C09135=1233.030,93.308,-46.941,-178.457,5.464,148.489
C09136=1233.025,93.557,-46.959,-178.455,5.465,148.489
C09137=1233.020,93.807,-46.977,-178.453,5.466,148.488
C09138=1233.016,94.056,-46.996,-178.450,5.466,148.487
C09139=1233.011,94.305,-47.014,-178.448,5.467,148.487
C09140=1233.006,94.555,-47.032,-178.445,5.468,148.486
C09141=1233.001,94.804,-47.052,-178.442,5.469,148.486
C09142=1232.996,95.053,-47.070,-178.439,5.470,148.485
C09143=1232.991,95.302,-47.088,-178.437,5.471,148.485
C09144=1232.986,95.552,-47.107,-178.435,5.471,148.484
C09145=1232.982,95.801,-47.126,-178.432,5.472,148.483
C09146=1232.976,96.050,-47.145,-178.429,5.473,148.483
C09147=1232.972,96.299,-47.164,-178.427,5.474,148.482
C09148=1232.967,96.549,-47.182,-178.425,5.474,148.482
C09149=1232.962,96.799,-47.201,-178.422,5.475,148.481
C09150=1232.958,97.047,-47.219,-178.420,5.476,148.481
C09151=1232.953,97.296,-47.237,-178.417,5.477,148.480
C09152=1232.948,97.546,-47.257,-178.414,5.478,148.479
C09153=1232.943,97.795,-47.275,-178.412,5.478,148.479
C09154=1232.938,98.044,-47.294,-178.409,5.479,148.478
C09155=1232.934,98.293,-47.313,-178.407,5.480,148.478
C09156=1232.928,98.543,-47.332,-178.404,5.481,148.477
C09157=1232.924,98.792,-47.351,-178.402,5.481,148.476
C09158=1232.919,99.041,-47.369,-178.399,5.482,148.476
C09159=1232.914,99.290,-47.388,-178.396,5.484,148.475
C09160=1232.909,99.540,-47.407,-178.394,5.484,148.475
C09161=1232.904,99.789,-47.426,-178.392,5.485,148.474
C09162=1232.900,100.038,-47.445,-178.389,5.486,148.473
C09163=1232.894,100.288,-47.464,-178.386,5.486,148.473
C09164=1232.890,100.537,-47.483,-178.384,5.487,148.472
C09165=1232.885,100.786,-47.501,-178.382,5.488,148.472
C09166=1232.880,101.035,-47.520,-178.379,5.489,148.471
C09167=1232.875,101.284,-47.539,-178.376,5.490,148.470
C09168=1232.871,101.534,-47.557,-178.374,5.491,148.470
C09169=1232.866,101.783,-47.577,-178.371,5.492,148.469
C09170=1232.861,102.032,-47.596,-178.368,5.492,148.469
C09171=1232.856,102.282,-47.615,-178.366,5.493,148.468
C09172=1232.852,102.531,-47.633,-178.364,5.494,148.468
C09173=1232.847,102.780,-47.653,-178.361,5.495,148.467
C09174=1232.842,103.029,-47.671,-178.358,5.496,148.466
C09175=1232.837,103.278,-47.690,-178.356,5.497,148.466
C09176=1232.832,103.527,-47.709,-178.353,5.498,148.465
C09177=1232.827,103.776,-47.729,-178.351,5.498,148.465
C09178=1232.823,104.026,-47.747,-178.348,5.499,148.464
C09179=1232.817,104.275,-47.766,-178.346,5.500,148.464
C09180=1232.813,104.525,-47.786,-178.343,5.500,148.463
C09181=1232.808,104.773,-47.805,-178.340,5.502,148.463
C09182=1232.803,105.023,-47.824,-178.338,5.503,148.462
C09183=1232.798,105.272,-47.842,-178.335,5.503,148.461
C09184=1232.794,105.521,-47.862,-178.333,5.504,148.461
C09185=1232.788,105.770,-47.881,-178.331,5.505,148.460
C09186=1232.784,106.020,-47.900,-178.328,5.506,148.460
C09187=1232.779,106.269,-47.919,-178.325,5.507,148.459
C09188=1232.775,106.518,-47.938,-178.323,5.508,148.459
C09189=1232.769,106.767,-47.957,-178.320,5.509,148.458
C09190=1232.765,107.017,-47.977,-178.318,5.510,148.457
C09191=1232.761,107.266,-47.996,-178.315,5.510,148.457
C09192=1232.755,107.534,-48.017,-178.312,5.512,148.456
C09193=1232.750,107.803,-48.037,-178.309,5.512,148.456
C09194=1232.744,108.071,-48.058,-178.307,5.513,148.455
C09195=1232.739,108.340,-48.079,-178.304,5.514,148.454
C09196=1232.734,108.589,-48.098,-178.302,5.515,148.454
C09197=1232.730,108.838,-48.117,-178.299,5.516,148.453
C09198=1232.725,109.087,-48.137,-178.296,5.517,148.453
C09199=1232.720,109.337,-48.155,-178.294,5.518,148.452
C09200=1232.716,109.586,-48.175,-178.292,5.518,148.452
C09201=1232.710,109.835,-48.194,-178.288,5.520,148.451
C09202=1232.706,110.085,-48.213,-178.286,5.521,148.451
C09203=1232.701,110.333,-48.232,-178.284,5.521,148.450
C09204=1232.696,110.583,-48.252,-178.281,5.522,148.449
C09205=1232.692,110.832,-48.272,-178.279,5.523,148.449
C09206=1232.686,111.081,-48.291,-178.276,5.524,148.448
C09207=1232.682,111.330,-48.310,-178.273,5.525,148.448
C09208=1232.677,111.579,-48.329,-178.271,5.526,148.447
C09209=1232.672,111.829,-48.349,-178.268,5.527,148.446
C09210=1232.667,112.079,-48.368,-178.266,5.527,148.446
C09211=1232.663,112.327,-48.387,-178.264,5.528,148.445
C09212=1232.658,112.577,-48.407,-178.261,5.530,148.445
C09213=1232.653,112.825,-48.426,-178.258,5.531,148.444
C09214=1232.648,113.074,-48.446,-178.256,5.531,148.444
C09215=1232.644,113.324,-48.466,-178.253,5.532,148.443
C09216=1232.639,113.573,-48.485,-178.251,5.533,148.443
C09217=1232.634,113.822,-48.504,-178.248,5.534,148.442
C09218=1232.629,114.072,-48.524,-178.245,5.535,148.441
C09219=1232.624,114.321,-48.543,-178.243,5.536,148.441
C09220=1232.619,114.570,-48.563,-178.241,5.536,148.440
C09221=1232.615,114.819,-48.582,-178.238,5.537,148.440
C09222=1232.610,115.068,-48.601,-178.235,5.539,148.439
C09223=1232.606,115.317,-48.622,-178.233,5.540,148.439
C09224=1232.600,115.566,-48.641,-178.231,5.541,148.438
C09225=1232.595,115.816,-48.661,-178.228,5.541,148.438
C09226=1232.591,116.065,-48.680,-178.225,5.543,148.437
C09227=1232.585,116.314,-48.700,-178.223,5.544,148.437
C09228=1232.581,116.563,-48.719,-178.220,5.544,148.436
C09229=1232.577,116.812,-48.739,-178.217,5.545,148.435
C09230=1232.572,117.062,-48.759,-178.215,5.546,148.435
C09231=1232.567,117.311,-48.778,-178.212,5.547,148.434
C09232=1232.562,117.560,-48.798,-178.210,5.548,148.434
C09233=1232.557,117.810,-48.817,-178.207,5.549,148.433
C09234=1232.552,118.058,-48.837,-178.205,5.549,148.433
C09235=1232.548,118.308,-48.857,-178.202,5.551,148.432
C09236=1232.543,118.557,-48.877,-178.199,5.552,148.432
C09237=1232.538,118.805,-48.897,-178.197,5.553,148.431
C09238=1232.534,119.055,-48.916,-178.195,5.554,148.431
C09239=1232.529,119.304,-48.935,-178.192,5.554,148.430
C09240=1232.524,119.554,-48.955,-178.189,5.556,148.429
C09241=1232.519,119.802,-48.975,-178.187,5.557,148.429
C09242=1232.515,120.052,-48.995,-178.184,5.557,148.428
C09243=1232.510,120.301,-49.014,-178.182,5.558,148.428
C09244=1232.505,120.550,-49.035,-178.179,5.560,148.427
C09245=1232.500,120.799,-49.054,-178.177,5.561,148.427
C09246=1232.495,121.049,-49.074,-178.174,5.561,148.426
C09247=1232.491,121.298,-49.094,-178.172,5.562,148.425
C09248=1232.486,121.547,-49.114,-178.169,5.564,148.425
C09249=1232.481,121.795,-49.134,-178.166,5.564,148.424
C09250=1232.476,122.045,-49.153,-178.164,5.565,148.424
C09251=1232.472,122.295,-49.173,-178.162,5.566,148.423
C09252=1232.467,122.543,-49.193,-178.158,5.567,148.423
C09253=1232.462,122.792,-49.213,-178.156,5.568,148.422
C09254=1232.457,123.041,-49.233,-178.154,5.569,148.422
C09255=1232.453,123.291,-49.253,-178.152,5.570,148.421
C09256=1232.448,123.540,-49.272,-178.148,5.571,148.421
C09257=1232.443,123.789,-49.293,-178.146,5.572,148.420
C09258=1232.438,124.038,-49.312,-178.144,5.573,148.420
C09259=1232.433,124.288,-49.333,-178.141,5.574,148.419
C09260=1232.428,124.537,-49.353,-178.138,5.576,148.419
C09261=1232.424,124.786,-49.373,-178.136,5.576,148.418
C09262=1232.419,125.036,-49.393,-178.133,5.577,148.417
C09263=1232.414,125.284,-49.413,-178.131,5.578,148.417
C09264=1232.409,125.533,-49.432,-178.128,5.579,148.416
C09265=1232.405,125.782,-49.453,-178.126,5.580,148.416
C09266=1232.400,126.032,-49.472,-178.123,5.581,148.415
C09267=1232.396,126.281,-49.493,-178.121,5.583,148.415
C09268=1232.391,126.530,-49.513,-178.118,5.583,148.414
C09269=1232.385,126.779,-49.533,-178.115,5.584,148.414
C09270=1232.381,127.028,-49.553,-178.113,5.585,148.413
C09271=1232.376,127.278,-49.573,-178.110,5.586,148.413
C09272=1232.371,127.526,-49.593,-178.108,5.587,148.412
C09273=1232.367,127.775,-49.614,-178.105,5.588,148.412
C09274=1232.362,128.025,-49.633,-178.103,5.589,148.411
C09275=1232.358,128.274,-49.654,-178.100,5.590,148.411
C09276=1232.352,128.524,-49.674,-178.097,5.591,148.410
C09277=1232.347,128.772,-49.694,-178.095,5.592,148.410
C09278=1232.343,129.021,-49.714,-178.092,5.594,148.409
C09279=1232.338,129.271,-49.734,-178.090,5.595,148.409
C09280=1232.334,129.520,-49.755,-178.087,5.595,148.408
C09281=1232.329,129.769,-49.775,-178.085,5.596,148.407
C09282=1232.324,130.018,-49.795,-178.082,5.598,148.407
C09283=1232.319,130.267,-49.816,-178.080,5.599,148.406
C09284=1232.315,130.516,-49.836,-178.077,5.599,148.406
C09285=1232.310,130.765,-49.856,-178.074,5.601,148.405
C09286=1232.304,131.014,-49.876,-178.072,5.602,148.405
C09287=1232.300,131.263,-49.897,-178.070,5.602,148.404
C09288=1232.295,131.512,-49.917,-178.067,5.604,148.404
C09289=1232.291,131.762,-49.937,-178.064,5.605,148.403
C09290=1232.286,132.011,-49.958,-178.062,5.606,148.403
C09291=1232.281,132.260,-49.978,-178.060,5.606,148.402
C09292=1232.277,132.509,-49.998,-178.057,5.608,148.402
C09293=1232.272,132.758,-50.019,-178.054,5.609,148.401
C09294=1232.267,133.008,-50.039,-178.052,5.610,148.400
C09295=1232.262,133.257,-50.059,-178.049,5.611,148.400
C09296=1232.257,133.525,-50.082,-178.046,5.612,148.399
C09297=1232.251,133.794,-50.103,-178.043,5.613,148.399
C09298=1232.247,134.063,-50.125,-178.041,5.614,148.398
C09299=1232.242,134.331,-50.148,-178.038,5.616,148.398
C09300=1232.237,134.581,-50.168,-178.035,5.617,148.397
C09301=1232.232,134.830,-50.189,-178.033,5.618,148.397
C09302=1232.228,135.079,-50.209,-178.030,5.619,148.396
C09303=1232.223,135.328,-50.229,-178.028,5.620,148.396
C09304=1232.218,135.577,-50.250,-178.025,5.621,148.395
C09305=1232.214,135.826,-50.271,-178.023,5.622,148.395
C09306=1232.209,136.075,-50.291,-178.020,5.623,148.394
C09307=1232.204,136.324,-50.312,-178.018,5.624,148.394
C09308=1232.200,136.573,-50.332,-178.015,5.626,148.393
C09309=1232.194,136.823,-50.353,-178.013,5.627,148.393
C09310=1232.190,137.071,-50.374,-178.010,5.627,148.392
C09311=1232.185,137.321,-50.393,-178.008,5.629,148.392
C09312=1232.180,137.570,-50.414,-178.005,5.630,148.391
C09313=1232.176,137.819,-50.435,-178.003,5.631,148.391
C09314=1232.170,138.069,-50.456,-178.000,5.632,148.390
C09315=1232.166,138.317,-50.476,-177.998,5.633,148.390
C09316=1232.161,138.567,-50.497,-177.995,5.634,148.389
C09317=1232.156,138.816,-50.517,-177.992,5.636,148.389
C09318=1232.152,139.065,-50.538,-177.990,5.636,148.388
C09319=1232.147,139.313,-50.559,-177.988,5.637,148.388
C09320=1232.143,139.562,-50.580,-177.984,5.639,148.387
C09321=1232.137,139.811,-50.601,-177.982,5.640,148.387
C09322=1232.133,140.060,-50.621,-177.980,5.640,148.386
C09323=1232.128,140.310,-50.642,-177.977,5.642,148.386
C09324=1232.123,140.559,-50.662,-177.974,5.643,148.385
C09325=1232.118,140.808,-50.683,-177.972,5.644,148.385
C09326=1232.114,141.057,-50.704,-177.969,5.645,148.384
C09327=1232.109,141.307,-50.725,-177.967,5.646,148.384
C09328=1232.105,141.556,-50.745,-177.964,5.647,148.383
C09329=1232.100,141.805,-50.766,-177.962,5.649,148.383
C09330=1232.095,142.053,-50.788,-177.959,5.649,148.382
C09331=1232.090,142.303,-50.808,-177.957,5.651,148.382
C09332=1232.086,142.552,-50.829,-177.954,5.652,148.381
C09333=1232.081,142.801,-50.850,-177.952,5.653,148.381
C09334=1232.076,143.050,-50.870,-177.949,5.654,148.380
C09335=1232.071,143.299,-50.891,-177.947,5.655,148.380
C09336=1232.067,143.547,-50.912,-177.944,5.656,148.379
C09337=1232.062,143.797,-50.934,-177.941,5.658,148.379
C09338=1232.057,144.047,-50.955,-177.939,5.658,148.378
C09339=1232.053,144.296,-50.975,-177.936,5.660,148.378
C09340=1232.048,144.545,-50.996,-177.933,5.661,148.377
C09341=1232.043,144.793,-51.017,-177.931,5.662,148.377
C09342=1232.038,145.042,-51.038,-177.928,5.663,148.376
C09343=1232.033,145.292,-51.059,-177.926,5.664,148.376
C09344=1232.030,145.541,-51.080,-177.923,5.665,148.375
C09345=1232.024,145.790,-51.101,-177.921,5.667,148.375
C09346=1232.020,146.039,-51.122,-177.919,5.668,148.374
C09347=1232.015,146.288,-51.143,-177.916,5.669,148.374
C09348=1232.010,146.537,-51.164,-177.913,5.670,148.373
C09349=1232.005,146.786,-51.185,-177.911,5.671,148.372
C09350=1232.001,147.036,-51.206,-177.908,5.673,148.372
C09351=1231.996,147.284,-51.228,-177.906,5.673,148.371
C09352=1231.992,147.533,-51.248,-177.903,5.675,148.371
C09353=1231.986,147.783,-51.269,-177.900,5.676,148.370
C09354=1231.982,148.031,-51.291,-177.898,5.677,148.370
C09355=1231.977,148.280,-51.311,-177.895,5.678,148.369
C09356=1231.973,148.529,-51.333,-177.893,5.679,148.369
C09357=1231.968,148.779,-51.354,-177.890,5.681,148.368
C09358=1231.963,149.028,-51.375,-177.888,5.682,148.368
C09359=1231.958,149.276,-51.396,-177.886,5.683,148.368
C09360=1231.953,149.526,-51.417,-177.882,5.684,148.367
C09361=1231.949,149.775,-51.439,-177.880,5.685,148.367
C09362=1231.944,150.024,-51.460,-177.877,5.687,148.366
C09363=1231.940,150.272,-51.481,-177.875,5.688,148.366
C09364=1231.934,150.522,-51.502,-177.873,5.688,148.365
C09365=1231.931,150.771,-51.523,-177.870,5.690,148.365
C09366=1231.926,151.020,-51.545,-177.867,5.691,148.364
C09367=1231.921,151.269,-51.566,-177.865,5.693,148.364
C09368=1231.916,151.518,-51.587,-177.862,5.694,148.363
C09369=1231.911,151.768,-51.609,-177.860,5.694,148.363
C09370=1231.907,152.016,-51.630,-177.857,5.696,148.362
C09371=1231.902,152.265,-51.651,-177.855,5.697,148.362
C09372=1231.897,152.514,-51.672,-177.852,5.699,148.361
C09373=1231.893,152.763,-51.694,-177.849,5.699,148.361
C09374=1231.887,153.013,-51.715,-177.847,5.701,148.360
C09375=1231.883,153.261,-51.736,-177.845,5.702,148.360
C09376=1231.878,153.510,-51.757,-177.842,5.703,148.359
C09377=1231.874,153.760,-51.779,-177.839,5.705,148.359
C09378=1231.869,154.008,-51.801,-177.837,5.705,148.358
C09379=1231.864,154.258,-51.822,-177.834,5.707,148.358
C09380=1231.860,154.507,-51.844,-177.832,5.708,148.357
C09381=1231.855,154.756,-51.865,-177.829,5.710,148.357
C09382=1231.850,155.004,-51.886,-177.827,5.711,148.357
C09383=1231.845,155.253,-51.908,-177.824,5.712,148.356
C09384=1231.841,155.503,-51.929,-177.822,5.713,148.356
C09385=1231.836,155.752,-51.951,-177.819,5.714,148.355
C09386=1231.831,156.000,-51.973,-177.816,5.716,148.355
C09387=1231.827,156.250,-51.994,-177.814,5.717,148.354
C09388=1231.822,156.499,-52.016,-177.811,5.718,148.354
C09389=1231.818,156.747,-52.037,-177.809,5.719,148.353
C09390=1231.813,156.997,-52.058,-177.806,5.721,148.353
C09391=1231.808,157.246,-52.080,-177.804,5.722,148.352
C09392=1231.803,157.495,-52.101,-177.801,5.723,148.352
C09393=1231.799,157.744,-52.123,-177.798,5.724,148.351
C09394=1231.794,157.993,-52.144,-177.796,5.725,148.351
C09395=1231.789,158.242,-52.166,-177.793,5.727,148.350
C09396=1231.785,158.491,-52.188,-177.791,5.728,148.350
C09397=1231.780,158.740,-52.210,-177.788,5.729,148.349
C09398=1231.776,158.989,-52.232,-177.786,5.730,148.349
C09399=1231.770,159.238,-52.253,-177.783,5.732,148.348
C09400=1231.765,159.507,-52.277,-177.781,5.733,148.348
C09401=1231.760,159.776,-52.300,-177.778,5.734,148.347
C09402=1231.755,160.046,-52.323,-177.775,5.736,148.347
C09403=1231.750,160.314,-52.347,-177.772,5.737,148.346
C09404=1231.746,160.563,-52.369,-177.770,5.738,148.346
C09405=1231.741,160.812,-52.390,-177.767,5.739,148.346
C09406=1231.736,161.062,-52.412,-177.764,5.741,148.345
C09407=1231.731,161.311,-52.434,-177.762,5.742,148.345
C09408=1231.726,161.559,-52.456,-177.760,5.744,148.344
C09409=1231.722,161.809,-52.478,-177.757,5.744,148.344
C09410=1231.717,162.057,-52.499,-177.754,5.746,148.343
C09411=1231.713,162.307,-52.521,-177.752,5.747,148.343
C09412=1231.708,162.555,-52.543,-177.749,5.749,148.342
C09413=1231.703,162.804,-52.565,-177.747,5.750,148.342
C09414=1231.699,163.053,-52.587,-177.744,5.751,148.341
C09415=1231.694,163.302,-52.608,-177.742,5.752,148.341
C09416=1231.690,163.551,-52.630,-177.739,5.754,148.340
C09417=1231.685,163.800,-52.652,-177.736,5.755,148.340
C09418=1231.681,164.049,-52.674,-177.734,5.757,148.339
C09419=1231.676,164.298,-52.696,-177.731,5.757,148.339
C09420=1231.671,164.547,-52.718,-177.729,5.759,148.339
C09421=1231.666,164.796,-52.740,-177.726,5.760,148.338
C09422=1231.662,165.046,-52.762,-177.723,5.762,148.338
C09423=1231.657,165.294,-52.784,-177.721,5.763,148.337
C09424=1231.652,165.544,-52.806,-177.719,5.764,148.337
C09425=1231.648,165.792,-52.828,-177.716,5.765,148.336
C09426=1231.643,166.042,-52.850,-177.713,5.767,148.336
C09427=1231.638,166.290,-52.871,-177.711,5.768,148.335
C09428=1231.633,166.539,-52.894,-177.708,5.769,148.335
C09429=1231.629,166.789,-52.916,-177.706,5.770,148.334
C09430=1231.624,167.038,-52.938,-177.703,5.772,148.334
C09431=1231.619,167.287,-52.959,-177.701,5.773,148.333
C09432=1231.615,167.535,-52.982,-177.698,5.775,148.333
C09433=1231.611,167.784,-53.004,-177.696,5.776,148.333
C09434=1231.606,168.034,-53.027,-177.693,5.777,148.332
C09435=1231.601,168.282,-53.048,-177.691,5.778,148.332
C09436=1231.596,168.532,-53.070,-177.688,5.780,148.331
C09437=1231.592,168.780,-53.092,-177.685,5.781,148.331
C09438=1231.587,169.029,-53.115,-177.683,5.783,148.330
C09439=1231.582,169.278,-53.137,-177.681,5.784,148.330
C09440=1231.578,169.527,-53.159,-177.678,5.785,148.329
C09441=1231.573,169.776,-53.181,-177.675,5.787,148.329
C09442=1231.568,170.025,-53.203,-177.673,5.788,148.329
C09443=1231.563,170.273,-53.226,-177.670,5.789,148.328
C09444=1231.559,170.523,-53.248,-177.668,5.790,148.328
C09445=1231.555,170.772,-53.270,-177.665,5.792,148.327
C09446=1231.549,171.021,-53.292,-177.662,5.793,148.327
C09447=1231.545,171.270,-53.315,-177.660,5.795,148.326
C09448=1231.540,171.518,-53.337,-177.658,5.796,148.326
C09449=1231.535,171.768,-53.359,-177.654,5.797,148.325
C09450=1231.531,172.016,-53.382,-177.652,5.798,148.325
C09451=1231.527,172.266,-53.404,-177.650,5.800,148.325
C09452=1231.522,172.515,-53.426,-177.647,5.801,148.324
C09453=1231.517,172.763,-53.449,-177.645,5.803,148.324
C09454=1231.513,173.013,-53.471,-177.642,5.805,148.323
C09455=1231.507,173.261,-53.493,-177.639,5.805,148.323
C09456=1231.503,173.510,-53.516,-177.637,5.807,148.322
C09457=1231.499,173.760,-53.538,-177.635,5.808,148.322
C09458=1231.493,174.008,-53.560,-177.632,5.810,148.322
C09459=1231.489,174.257,-53.583,-177.629,5.811,148.321
C09460=1231.485,174.507,-53.605,-177.627,5.812,148.321
C09461=1231.480,174.755,-53.628,-177.625,5.813,148.320
C09462=1231.475,175.004,-53.650,-177.621,5.815,148.320
C09463=1231.470,175.253,-53.672,-177.619,5.817,148.319
C09464=1231.466,175.502,-53.695,-177.617,5.818,148.319
C09465=1231.462,175.751,-53.717,-177.614,5.819,148.318
C09466=1231.456,176.000,-53.740,-177.611,5.820,148.318
C09467=1231.452,176.249,-53.762,-177.609,5.822,148.318
C09468=1231.447,176.498,-53.786,-177.607,5.823,148.317
C09469=1231.442,176.747,-53.807,-177.604,5.825,148.317
C09470=1231.438,176.996,-53.831,-177.601,5.826,148.316
C09471=1231.433,177.245,-53.853,-177.599,5.827,148.316
C09472=1231.428,177.493,-53.876,-177.596,5.829,148.315
C09473=1231.424,177.743,-53.898,-177.594,5.830,148.315
C09474=1231.420,177.991,-53.920,-177.591,5.832,148.315
C09475=1231.415,178.241,-53.943,-177.588,5.834,148.314
C09476=1231.410,178.489,-53.965,-177.586,5.834,148.314
C09477=1231.406,178.738,-53.989,-177.583,5.836,148.313
C09478=1231.401,178.987,-54.011,-177.581,5.837,148.313
C09479=1231.396,179.236,-54.034,-177.578,5.839,148.312
C09480=1231.392,179.485,-54.056,-177.576,5.840,148.312
C09481=1231.387,179.734,-54.079,-177.573,5.842,148.312
C09482=1231.382,179.982,-54.102,-177.570,5.843,148.311
C09483=1231.378,180.232,-54.124,-177.568,5.844,148.311
C09484=1231.373,180.481,-54.148,-177.565,5.846,148.310
C09485=1231.369,180.730,-54.170,-177.563,5.847,148.310
C09486=1231.363,180.978,-54.193,-177.561,5.849,148.310
C09487=1231.359,181.227,-54.215,-177.557,5.850,148.309
C09488=1231.355,181.476,-54.239,-177.555,5.851,148.309
C09489=1231.350,181.726,-54.261,-177.553,5.853,148.308
C09490=1231.345,181.974,-54.284,-177.551,5.854,148.308
C09491=1231.340,182.223,-54.307,-177.547,5.856,148.307
C09492=1231.336,182.472,-54.329,-177.545,5.858,148.307
C09493=1231.331,182.721,-54.353,-177.543,5.859,148.307
C09494=1231.327,182.970,-54.375,-177.540,5.860,148.306
C09495=1231.322,183.218,-54.398,-177.537,5.862,148.306
C09496=1231.317,183.468,-54.421,-177.535,5.863,148.305
C09497=1231.313,183.717,-54.444,-177.532,5.865,148.305
C09498=1231.308,183.966,-54.467,-177.530,5.866,148.304
C09499=1231.304,184.214,-54.490,-177.527,5.867,148.304
C09500=1231.299,184.463,-54.513,-177.524,5.869,148.304
C09501=1231.294,184.712,-54.536,-177.522,5.870,148.303
C09502=1231.290,184.961,-54.558,-177.520,5.872,148.303
C09503=1231.286,185.210,-54.582,-177.516,5.874,148.302
C09504=1231.280,185.480,-54.607,-177.514,5.875,148.302
C09505=1231.276,185.749,-54.631,-177.512,5.876,148.302
C09506=1231.270,186.019,-54.656,-177.509,5.878,148.301
C09507=1231.265,186.289,-54.681,-177.506,5.880,148.301
C09508=1231.261,186.538,-54.704,-177.503,5.881,148.300
C09509=1231.256,186.787,-54.727,-177.501,5.882,148.300
C09510=1231.251,187.035,-54.750,-177.498,5.884,148.299
C09511=1231.246,187.284,-54.774,-177.496,5.885,148.299
C09512=1231.242,187.533,-54.796,-177.493,5.887,148.299
C09513=1231.238,187.782,-54.820,-177.490,5.889,148.298
C09514=1231.233,188.031,-54.843,-177.488,5.890,148.298
C09515=1231.228,188.280,-54.867,-177.485,5.891,148.297
C09516=1231.224,188.529,-54.889,-177.483,5.893,148.297
C09517=1231.220,188.778,-54.913,-177.480,5.894,148.296
C09518=1231.214,189.026,-54.936,-177.478,5.896,148.296
C09519=1231.210,189.275,-54.959,-177.475,5.898,148.296
C09520=1231.206,189.524,-54.982,-177.473,5.899,148.295
C09521=1231.201,189.773,-55.005,-177.470,5.900,148.295
C09522=1231.196,190.022,-55.028,-177.467,5.902,148.294
C09523=1231.192,190.271,-55.052,-177.465,5.903,148.294
C09524=1231.187,190.520,-55.075,-177.462,5.905,148.294
C09525=1231.182,190.769,-55.099,-177.460,5.907,148.293
C09526=1231.178,191.018,-55.121,-177.458,5.908,148.293
C09527=1231.173,191.266,-55.144,-177.455,5.909,148.292
C09528=1231.168,191.515,-55.168,-177.452,5.911,148.292
C09529=1231.164,191.764,-55.191,-177.450,5.912,148.292
C09530=1231.159,192.013,-55.214,-177.447,5.914,148.291
C09531=1231.154,192.261,-55.238,-177.445,5.916,148.291
C09532=1231.150,192.510,-55.262,-177.442,5.917,148.290
C09533=1231.146,192.759,-55.285,-177.439,5.918,148.290
C09534=1231.141,193.008,-55.308,-177.437,5.920,148.290
C09535=1231.136,193.257,-55.331,-177.435,5.921,148.289
C09536=1231.132,193.506,-55.355,-177.432,5.923,148.289
C09537=1231.127,193.755,-55.379,-177.429,5.925,148.288
C09538=1231.123,194.004,-55.402,-177.427,5.926,148.288
C09539=1231.118,194.253,-55.425,-177.424,5.927,148.288
C09540=1231.113,194.502,-55.449,-177.421,5.929,148.287
C09541=1231.108,194.751,-55.472,-177.419,5.930,148.287
C09542=1231.104,194.999,-55.496,-177.417,5.932,148.286
C09543=1231.099,195.248,-55.520,-177.414,5.934,148.286
C09544=1231.095,195.497,-55.543,-177.411,5.936,148.286
C09545=1231.090,195.746,-55.566,-177.409,5.937,148.285
C09546=1231.086,195.995,-55.590,-177.406,5.938,148.285
C09547=1231.082,196.244,-55.613,-177.404,5.940,148.285
C09548=1231.077,196.493,-55.637,-177.402,5.941,148.284
C09549=1231.073,196.741,-55.661,-177.398,5.943,148.284
C09550=1231.068,196.990,-55.684,-177.396,5.945,148.283
C09551=1231.063,197.239,-55.707,-177.394,5.946,148.283
C09552=1231.059,197.487,-55.731,-177.391,5.948,148.283
C09553=1231.054,197.736,-55.755,-177.388,5.949,148.282
C09554=1231.049,197.986,-55.779,-177.386,5.951,148.282
C09555=1231.044,198.234,-55.803,-177.383,5.952,148.281
C09556=1231.039,198.483,-55.826,-177.381,5.954,148.281
C09557=1231.035,198.732,-55.849,-177.378,5.956,148.281
C09558=1231.030,198.981,-55.874,-177.376,5.957,148.280
C09559=1231.026,199.230,-55.897,-177.373,5.959,148.280
C09560=1231.021,199.478,-55.921,-177.371,5.960,148.280
C09561=1231.017,199.727,-55.944,-177.367,5.962,148.279
C09562=1231.012,199.976,-55.968,-177.365,5.963,148.279
C09563=1231.008,200.225,-55.992,-177.363,5.965,148.278
C09564=1231.003,200.474,-56.015,-177.360,5.967,148.278
C09565=1230.998,200.722,-56.039,-177.357,5.969,148.278
C09566=1230.994,200.971,-56.063,-177.355,5.970,148.277
C09567=1230.990,201.220,-56.087,-177.353,5.971,148.277
C09568=1230.984,201.470,-56.111,-177.350,5.973,148.276
C09569=1230.980,201.718,-56.135,-177.348,5.974,148.276
C09570=1230.975,201.967,-56.158,-177.345,5.976,148.276
C09571=1230.971,202.215,-56.182,-177.342,5.978,148.275
C09572=1230.967,202.464,-56.207,-177.340,5.980,148.275
C09573=1230.962,202.713,-56.230,-177.338,5.981,148.274
C09574=1230.958,202.961,-56.254,-177.335,5.982,148.274
C09575=1230.952,203.211,-56.278,-177.332,5.984,148.274
C09576=1230.948,203.460,-56.302,-177.329,5.986,148.273
C09577=1230.944,203.709,-56.326,-177.327,5.987,148.273
C09578=1230.939,203.957,-56.350,-177.324,5.989,148.273
C09579=1230.935,204.206,-56.374,-177.322,5.991,148.272
C09580=1230.929,204.455,-56.398,-177.319,5.992,148.272
C09581=1230.925,204.703,-56.422,-177.317,5.993,148.272
C09582=1230.921,204.952,-56.446,-177.314,5.995,148.271
C09583=1230.916,205.201,-56.470,-177.312,5.997,148.271
C09584=1230.912,205.450,-56.494,-177.309,5.999,148.270
C09585=1230.907,205.699,-56.518,-177.307,6.000,148.270
C09586=1230.902,205.948,-56.542,-177.304,6.002,148.270
C09587=1230.898,206.196,-56.566,-177.301,6.003,148.269
C09588=1230.893,206.444,-56.590,-177.299,6.005,148.269
C09589=1230.889,206.695,-56.614,-177.296,6.007,148.269
C09590=1230.884,206.943,-56.638,-177.294,6.008,148.268
C09591=1230.880,207.191,-56.662,-177.291,6.010,148.268
C09592=1230.875,207.440,-56.687,-177.289,6.012,148.268
C09593=1230.870,207.689,-56.710,-177.286,6.013,148.267
C09594=1230.866,207.938,-56.735,-177.284,6.014,148.267
C09595=1230.862,208.187,-56.759,-177.281,6.016,148.266
C09596=1230.857,208.435,-56.784,-177.278,6.018,148.266
C09597=1230.852,208.684,-56.808,-177.276,6.020,148.266
C09598=1230.848,208.933,-56.831,-177.274,6.021,148.265
C09599=1230.843,209.182,-56.856,-177.271,6.023,148.265
C09600=1230.839,209.431,-56.880,-177.268,6.025,148.265
C09601=1230.834,209.679,-56.904,-177.266,6.027,148.264
C09602=1230.829,209.928,-56.929,-177.263,6.029,148.264
C09603=1230.825,210.177,-56.953,-177.261,6.030,148.263
C09604=1230.820,210.426,-56.978,-177.258,6.031,148.263
C09605=1230.816,210.675,-57.001,-177.255,6.033,148.263
C09606=1230.811,210.923,-57.025,-177.253,6.035,148.262
C09607=1230.807,211.172,-57.051,-177.250,6.037,148.262
C09608=1230.801,211.443,-57.077,-177.247,6.039,148.262
C09609=1230.797,211.712,-57.103,-177.245,6.040,148.261
C09610=1230.792,211.983,-57.130,-177.242,6.042,148.261
C09611=1230.787,212.254,-57.156,-177.239,6.044,148.260
C09612=1230.783,212.503,-57.180,-177.236,6.046,148.260
C09613=1230.777,212.751,-57.205,-177.234,6.047,148.260
C09614=1230.773,213.000,-57.229,-177.232,6.049,148.259
C09615=1230.769,213.249,-57.254,-177.229,6.050,148.259
C09616=1230.764,213.498,-57.278,-177.226,6.052,148.259
C09617=1230.759,213.746,-57.303,-177.224,6.054,148.258
C09618=1230.755,213.995,-57.327,-177.222,6.055,148.258
C09619=1230.750,214.244,-57.352,-177.219,6.057,148.258
C09620=1230.746,214.493,-57.376,-177.216,6.059,148.257
C09621=1230.741,214.742,-57.401,-177.214,6.061,148.257
C09622=1230.737,214.990,-57.426,-177.211,6.062,148.256
C09623=1230.732,215.238,-57.451,-177.208,6.064,148.256
C09624=1230.728,215.488,-57.475,-177.206,6.065,148.256
C09625=1230.723,215.736,-57.500,-177.203,6.067,148.255
C09626=1230.719,215.985,-57.524,-177.201,6.069,148.255
C09627=1230.714,216.234,-57.549,-177.198,6.071,148.255
C09628=1230.710,216.483,-57.573,-177.196,6.073,148.254
C09629=1230.705,216.731,-57.598,-177.193,6.075,148.254
C09630=1230.701,216.980,-57.623,-177.191,6.076,148.254
C09631=1230.696,217.228,-57.647,-177.188,6.077,148.253
C09632=1230.691,217.477,-57.672,-177.186,6.079,148.253
C09633=1230.687,217.726,-57.697,-177.183,6.081,148.253
C09634=1230.682,217.975,-57.721,-177.180,6.083,148.252
C09635=1230.678,218.224,-57.746,-177.178,6.085,148.252
C09636=1230.673,218.472,-57.771,-177.176,6.086,148.252
C09637=1230.668,218.721,-57.796,-177.173,6.088,148.251
C09638=1230.664,218.970,-57.820,-177.170,6.090,148.251
C09639=1230.659,219.219,-57.845,-177.168,6.092,148.251
C09640=1230.656,219.467,-57.870,-177.165,6.093,148.250
C09641=1230.651,219.716,-57.895,-177.162,6.095,148.250
C09642=1230.645,219.965,-57.919,-177.160,6.097,148.250
C09643=1230.642,220.213,-57.945,-177.158,6.098,148.249
C09644=1230.637,220.462,-57.969,-177.155,6.100,148.249
C09645=1230.632,220.711,-57.994,-177.153,6.102,148.249
C09646=1230.628,220.959,-58.019,-177.150,6.104,148.248
C09647=1230.624,221.209,-58.044,-177.147,6.106,148.248
C09648=1230.619,221.457,-58.069,-177.145,6.108,148.248
C09649=1230.615,221.705,-58.094,-177.143,6.109,148.247
C09650=1230.610,221.955,-58.119,-177.140,6.110,148.247
C09651=1230.605,222.203,-58.143,-177.137,6.112,148.247
C09652=1230.601,222.452,-58.168,-177.135,6.114,148.246
C09653=1230.596,222.701,-58.193,-177.132,6.116,148.246
C09654=1230.592,222.949,-58.219,-177.129,6.118,148.246
C09655=1230.587,223.198,-58.243,-177.127,6.120,148.245
C09656=1230.583,223.447,-58.269,-177.125,6.121,148.245
C09657=1230.578,223.695,-58.293,-177.122,6.123,148.245
C09658=1230.574,223.945,-58.318,-177.120,6.125,148.244
C09659=1230.569,224.193,-58.344,-177.117,6.126,148.244
C09660=1230.565,224.442,-58.368,-177.114,6.128,148.244
C09661=1230.560,224.690,-58.394,-177.112,6.130,148.243
C09662=1230.556,224.939,-58.419,-177.109,6.132,148.243
C09663=1230.551,225.188,-58.444,-177.106,6.134,148.243
C09664=1230.546,225.437,-58.469,-177.104,6.135,148.242
C09665=1230.542,225.685,-58.494,-177.102,6.137,148.242
C09666=1230.538,225.934,-58.519,-177.099,6.139,148.242
C09667=1230.533,226.182,-58.544,-177.096,6.141,148.241
C09668=1230.529,226.431,-58.570,-177.094,6.142,148.241
C09669=1230.524,226.680,-58.595,-177.091,6.144,148.241
C09670=1230.519,226.929,-58.620,-177.089,6.146,148.241
C09671=1230.515,227.177,-58.644,-177.087,6.147,148.240
C09672=1230.511,227.426,-58.670,-177.084,6.149,148.240
C09673=1230.506,227.674,-58.696,-177.081,6.151,148.240
C09674=1230.501,227.923,-58.721,-177.079,6.153,148.239
C09675=1230.497,228.172,-58.746,-177.076,6.155,148.239
C09676=1230.492,228.420,-58.772,-177.073,6.157,148.239
C09677=1230.488,228.670,-58.797,-177.071,6.158,148.238
C09678=1230.483,228.918,-58.822,-177.068,6.160,148.238
C09679=1230.479,229.167,-58.848,-177.066,6.162,148.238
C09680=1230.474,229.415,-58.872,-177.064,6.163,148.237
C09681=1230.470,229.664,-58.898,-177.061,6.165,148.237
C09682=1230.466,229.913,-58.923,-177.059,6.167,148.237
C09683=1230.461,230.161,-58.948,-177.056,6.169,148.236
C09684=1230.457,230.410,-58.974,-177.054,6.171,148.236
C09685=1230.452,230.658,-58.999,-177.051,6.173,148.236
C09686=1230.447,230.907,-59.025,-177.048,6.175,148.236
C09687=1230.443,231.156,-59.050,-177.046,6.177,148.235
C09688=1230.438,231.405,-59.075,-177.043,6.179,148.235
C09689=1230.434,231.653,-59.101,-177.041,6.180,148.235
C09690=1230.429,231.901,-59.127,-177.038,6.181,148.234
C09691=1230.425,232.150,-59.152,-177.036,6.183,148.234
C09692=1230.420,232.400,-59.177,-177.033,6.185,148.234
C09693=1230.416,232.648,-59.203,-177.030,6.187,148.233
C09694=1230.411,232.897,-59.229,-177.028,6.189,148.233
C09695=1230.407,233.145,-59.254,-177.026,6.191,148.233
C09696=1230.402,233.394,-59.280,-177.023,6.193,148.233
C09697=1230.398,233.642,-59.305,-177.021,6.195,148.232
C09698=1230.394,233.891,-59.331,-177.018,6.197,148.232
C09699=1230.389,234.139,-59.357,-177.016,6.198,148.232
C09700=1230.384,234.389,-59.382,-177.013,6.200,148.231
C09701=1230.380,234.637,-59.407,-177.011,6.202,148.231
C09702=1230.375,234.886,-59.433,-177.008,6.203,148.231
C09703=1230.371,235.134,-59.458,-177.005,6.205,148.230
C09704=1230.366,235.384,-59.485,-177.003,6.207,148.230
C09705=1230.361,235.632,-59.510,-177.001,6.209,148.230
C09706=1230.357,235.880,-59.536,-176.998,6.211,148.230
C09707=1230.353,236.129,-59.562,-176.995,6.213,148.229
C09708=1230.348,236.377,-59.587,-176.993,6.215,148.229
C09709=1230.344,236.626,-59.613,-176.990,6.217,148.229
C09710=1230.340,236.875,-59.639,-176.988,6.219,148.228
C09711=1230.335,237.124,-59.664,-176.985,6.220,148.228
C09712=1230.330,237.395,-59.692,-176.982,6.223,148.228
C09713=1230.326,237.666,-59.721,-176.980,6.224,148.227
C09714=1230.320,237.938,-59.749,-176.977,6.226,148.227
C09715=1230.315,238.210,-59.777,-176.974,6.228,148.227
C09716=1230.311,238.458,-59.804,-176.972,6.230,148.226
C09717=1230.306,238.706,-59.829,-176.969,6.232,148.226
C09718=1230.302,238.955,-59.855,-176.967,6.234,148.226
C09719=1230.298,239.204,-59.880,-176.964,6.236,148.226
C09720=1230.293,239.453,-59.907,-176.962,6.238,148.225
C09721=1230.288,239.701,-59.932,-176.959,6.240,148.225
C09722=1230.284,239.950,-59.958,-176.957,6.242,148.225
C09723=1230.280,240.198,-59.984,-176.954,6.244,148.224
C09724=1230.276,240.447,-60.010,-176.951,6.245,148.224
C09725=1230.270,240.695,-60.036,-176.949,6.247,148.224
C09726=1230.266,240.944,-60.062,-176.947,6.249,148.224
C09727=1230.262,241.193,-60.088,-176.945,6.251,148.223
C09728=1230.257,241.441,-60.113,-176.942,6.252,148.223
C09729=1230.253,241.690,-60.140,-176.939,6.254,148.223
C09730=1230.248,241.938,-60.166,-176.937,6.256,148.222
C09731=1230.244,242.187,-60.192,-176.934,6.258,148.222
C09732=1230.239,242.436,-60.218,-176.932,6.260,148.222
C09733=1230.235,242.684,-60.244,-176.929,6.262,148.222
C09734=1230.231,242.933,-60.270,-176.927,6.264,148.221
C09735=1230.226,243.182,-60.296,-176.924,6.266,148.221
C09736=1230.221,243.429,-60.323,-176.922,6.268,148.221
C09737=1230.217,243.678,-60.348,-176.919,6.270,148.220
C09738=1230.213,243.927,-60.374,-176.917,6.272,148.220
C09739=1230.208,244.176,-60.401,-176.914,6.274,148.220
C09740=1230.204,244.424,-60.427,-176.912,6.276,148.220
C09741=1230.199,244.673,-60.453,-176.909,6.278,148.219
C09742=1230.194,244.921,-60.479,-176.906,6.279,148.219
C09743=1230.190,245.170,-60.505,-176.904,6.281,148.219
C09744=1230.185,245.419,-60.531,-176.902,6.283,148.219
C09745=1230.181,245.667,-60.558,-176.899,6.285,148.218
C09746=1230.177,245.916,-60.584,-176.896,6.287,148.218
C09747=1230.172,246.164,-60.611,-176.894,6.289,148.218
C09748=1230.168,246.413,-60.636,-176.891,6.291,148.217
C09749=1230.163,246.662,-60.664,-176.889,6.293,148.217
C09750=1230.159,246.910,-60.689,-176.886,6.295,148.217
C09751=1230.154,247.159,-60.715,-176.884,6.297,148.217
C09752=1230.150,247.407,-60.742,-176.881,6.299,148.216
C09753=1230.146,247.656,-60.767,-176.879,6.301,148.216
C09754=1230.141,247.904,-60.795,-176.877,6.302,148.216
C09755=1230.137,248.153,-60.820,-176.874,6.304,148.216
C09756=1230.132,248.402,-60.847,-176.872,6.306,148.215
C09757=1230.128,248.650,-60.874,-176.869,6.308,148.215
C09758=1230.123,248.899,-60.900,-176.867,6.310,148.215
C09759=1230.119,249.147,-60.927,-176.864,6.312,148.215
C09760=1230.114,249.396,-60.953,-176.862,6.314,148.214
C09761=1230.110,249.644,-60.979,-176.859,6.316,148.214
C09762=1230.105,249.893,-61.005,-176.857,6.318,148.214
C09763=1230.101,250.141,-61.032,-176.855,6.320,148.214
C09764=1230.096,250.390,-61.059,-176.852,6.322,148.213
C09765=1230.092,250.638,-61.085,-176.849,6.323,148.213
C09766=1230.087,250.887,-61.112,-176.847,6.325,148.213
C09767=1230.083,251.136,-61.138,-176.845,6.328,148.213
C09768=1230.078,251.384,-61.165,-176.842,6.329,148.212
C09769=1230.074,251.632,-61.191,-176.839,6.331,148.212
C09770=1230.070,251.881,-61.217,-176.837,6.333,148.212
C09771=1230.065,252.130,-61.244,-176.835,6.335,148.212
C09772=1230.061,252.378,-61.271,-176.832,6.337,148.211
C09773=1230.056,252.627,-61.298,-176.829,6.339,148.211
C09774=1230.052,252.875,-61.324,-176.827,6.341,148.211
C09775=1230.047,253.124,-61.351,-176.825,6.343,148.211
C09776=1230.043,253.372,-61.377,-176.822,6.345,148.210
C09777=1230.039,253.621,-61.404,-176.819,6.347,148.210
C09778=1230.034,253.870,-61.431,-176.817,6.349,148.210
C09779=1230.030,254.118,-61.457,-176.815,6.351,148.210
C09780=1230.025,254.366,-61.484,-176.812,6.354,148.209
C09781=1230.021,254.615,-61.511,-176.809,6.356,148.209
C09782=1230.016,254.864,-61.537,-176.806,6.358,148.209
C09783=1230.012,255.112,-61.564,-176.804,6.360,148.209
C09784=1230.007,255.361,-61.591,-176.802,6.362,148.208
C09785=1230.003,255.609,-61.618,-176.799,6.364,148.208
C09786=1229.999,255.857,-61.645,-176.797,6.366,148.208
C09787=1229.994,256.106,-61.672,-176.794,6.368,148.208
C09788=1229.990,256.355,-61.698,-176.792,6.370,148.207
C09789=1229.986,256.604,-61.725,-176.789,6.372,148.207
C09790=1229.981,256.852,-61.752,-176.787,6.374,148.207
C09791=1229.977,257.101,-61.778,-176.784,6.376,148.207
C09792=1229.972,257.349,-61.805,-176.782,6.378,148.206
C09793=1229.968,257.598,-61.833,-176.780,6.380,148.206
C09794=1229.963,257.846,-61.860,-176.777,6.382,148.206
C09795=1229.959,258.094,-61.886,-176.774,6.383,148.206
C09796=1229.954,258.343,-61.913,-176.772,6.385,148.205
C09797=1229.950,258.591,-61.940,-176.770,6.388,148.205
C09798=1229.945,258.840,-61.967,-176.767,6.389,148.205
C09799=1229.940,259.088,-61.994,-176.764,6.391,148.205
C09800=1229.937,259.337,-62.021,-176.762,6.394,148.205
C09801=1229.933,259.586,-62.048,-176.760,6.395,148.204
C09802=1229.928,259.834,-62.075,-176.757,6.397,148.204
C09803=1229.923,260.083,-62.102,-176.755,6.400,148.204
C09804=1229.919,260.331,-62.129,-176.752,6.401,148.204
C09805=1229.915,260.579,-62.156,-176.750,6.403,148.203
C09806=1229.910,260.828,-62.183,-176.747,6.406,148.203
C09807=1229.905,261.076,-62.210,-176.745,6.408,148.203
C09808=1229.901,261.325,-62.237,-176.742,6.410,148.203
C09809=1229.897,261.574,-62.264,-176.740,6.412,148.203
C09810=1229.892,261.822,-62.292,-176.737,6.414,148.202
C09811=1229.888,262.070,-62.319,-176.735,6.416,148.202
C09812=1229.884,262.318,-62.346,-176.732,6.418,148.202
C09813=1229.879,262.567,-62.373,-176.730,6.420,148.202
C09814=1229.875,262.816,-62.400,-176.727,6.422,148.201
C09815=1229.870,263.065,-62.427,-176.725,6.424,148.201
C09816=1229.866,263.337,-62.457,-176.723,6.426,148.201
C09817=1229.861,263.610,-62.487,-176.719,6.429,148.201
C09818=1229.856,263.882,-62.517,-176.717,6.431,148.200
C09819=1229.850,264.155,-62.547,-176.714,6.434,148.200
C09820=1229.846,264.403,-62.574,-176.712,6.436,148.200
C09821=1229.842,264.651,-62.601,-176.709,6.438,148.200
C09822=1229.838,264.900,-62.628,-176.707,6.440,148.200
C09823=1229.833,265.149,-62.655,-176.704,6.442,148.199
C09824=1229.829,265.397,-62.683,-176.702,6.444,148.199
C09825=1229.824,265.645,-62.710,-176.699,6.446,148.199
C09826=1229.820,265.894,-62.738,-176.697,6.448,148.199
C09827=1229.816,266.142,-62.765,-176.694,6.450,148.198
C09828=1229.811,266.391,-62.792,-176.692,6.452,148.198
C09829=1229.807,266.639,-62.820,-176.690,6.454,148.198
C09830=1229.803,266.888,-62.848,-176.687,6.457,148.198
C09831=1229.798,267.136,-62.875,-176.684,6.459,148.198
C09832=1229.794,267.385,-62.902,-176.682,6.461,148.197
C09833=1229.789,267.633,-62.930,-176.680,6.463,148.197
C09834=1229.785,267.882,-62.957,-176.677,6.465,148.197
C09835=1229.781,268.130,-62.985,-176.675,6.467,148.197
C09836=1229.776,268.378,-63.012,-176.672,6.469,148.197
C09837=1229.771,268.627,-63.040,-176.670,6.471,148.196
C09838=1229.767,268.876,-63.068,-176.668,6.473,148.196
C09839=1229.762,269.124,-63.095,-176.665,6.475,148.196
C09840=1229.758,269.372,-63.123,-176.662,6.478,148.196
C09841=1229.753,269.621,-63.150,-176.660,6.480,148.196
C09842=1229.750,269.869,-63.178,-176.657,6.482,148.195
C09843=1229.745,270.118,-63.205,-176.655,6.484,148.195
C09844=1229.741,270.366,-63.233,-176.652,6.486,148.195
C09845=1229.737,270.615,-63.260,-176.650,6.488,148.195
C09846=1229.732,270.863,-63.288,-176.648,6.490,148.195
C09847=1229.727,271.111,-63.315,-176.646,6.492,148.195
C09848=1229.723,271.360,-63.344,-176.643,6.494,148.194
C09849=1229.718,271.609,-63.371,-176.640,6.497,148.194
C09850=1229.714,271.856,-63.398,-176.638,6.499,148.194
C09851=1229.710,272.106,-63.426,-176.635,6.501,148.194
C09852=1229.706,272.353,-63.454,-176.633,6.503,148.194
C09853=1229.701,272.601,-63.481,-176.630,6.505,148.193
C09854=1229.697,272.851,-63.509,-176.628,6.507,148.193
C09855=1229.692,273.099,-63.537,-176.626,6.509,148.193
C09856=1229.688,273.347,-63.564,-176.624,6.511,148.193
C09857=1229.684,273.596,-63.592,-176.620,6.514,148.193
C09858=1229.679,273.844,-63.620,-176.618,6.516,148.193
C09859=1229.675,274.093,-63.648,-176.616,6.518,148.192
C09860=1229.670,274.341,-63.676,-176.614,6.520,148.192
C09861=1229.666,274.589,-63.704,-176.611,6.522,148.192
C09862=1229.662,274.838,-63.732,-176.609,6.524,148.192
C09863=1229.657,275.086,-63.760,-176.606,6.526,148.192
C09864=1229.652,275.334,-63.787,-176.603,6.529,148.191
C09865=1229.649,275.583,-63.815,-176.601,6.531,148.191
C09866=1229.644,275.831,-63.843,-176.598,6.533,148.191
C09867=1229.640,276.080,-63.871,-176.596,6.535,148.191
C09868=1229.635,276.328,-63.899,-176.594,6.537,148.191
C09869=1229.631,276.576,-63.927,-176.592,6.540,148.190
C09870=1229.626,276.825,-63.956,-176.589,6.541,148.190
C09871=1229.622,277.073,-63.983,-176.586,6.544,148.190
C09872=1229.618,277.322,-64.011,-176.584,6.546,148.190
C09873=1229.614,277.570,-64.039,-176.582,6.549,148.190
C09874=1229.609,277.819,-64.067,-176.579,6.551,148.190
C09875=1229.605,278.066,-64.095,-176.577,6.553,148.189
C09876=1229.601,278.315,-64.123,-176.575,6.555,148.189
C09877=1229.596,278.564,-64.151,-176.572,6.558,148.189
C09878=1229.591,278.812,-64.179,-176.570,6.560,148.189
C09879=1229.587,279.061,-64.207,-176.567,6.562,148.189
C09880=1229.582,279.309,-64.235,-176.565,6.564,148.189
C09881=1229.579,279.557,-64.263,-176.562,6.566,148.188
C09882=1229.574,279.805,-64.292,-176.560,6.568,148.188
C09883=1229.570,280.054,-64.320,-176.557,6.571,148.188
C09884=1229.566,280.302,-64.348,-176.555,6.573,148.188
C09885=1229.561,280.551,-64.376,-176.552,6.575,148.188
C09886=1229.557,280.798,-64.404,-176.550,6.577,148.188
C09887=1229.552,281.047,-64.433,-176.548,6.579,148.187
C09888=1229.548,281.295,-64.461,-176.545,6.581,148.187
C09889=1229.543,281.544,-64.489,-176.543,6.584,148.187
C09890=1229.539,281.792,-64.517,-176.540,6.586,148.187
C09891=1229.535,282.041,-64.545,-176.538,6.588,148.187
C09892=1229.530,282.289,-64.574,-176.535,6.590,148.187
C09893=1229.526,282.537,-64.602,-176.533,6.593,148.187
C09894=1229.521,282.786,-64.630,-176.531,6.594,148.186
C09895=1229.518,283.034,-64.658,-176.528,6.598,148.186
C09896=1229.513,283.283,-64.687,-176.526,6.600,148.186
C09897=1229.509,283.531,-64.715,-176.523,6.602,148.186
C09898=1229.504,283.780,-64.744,-176.521,6.604,148.186
C09899=1229.500,284.028,-64.771,-176.519,6.606,148.186
C09900=1229.496,284.276,-64.801,-176.516,6.609,148.186
C09901=1229.491,284.524,-64.829,-176.514,6.611,148.186
C09902=1229.487,284.773,-64.857,-176.511,6.613,148.185
C09903=1229.483,285.021,-64.885,-176.509,6.615,148.185
C09904=1229.478,285.269,-64.914,-176.507,6.617,148.185
C09905=1229.474,285.518,-64.943,-176.504,6.620,148.185
C09906=1229.469,285.766,-64.971,-176.502,6.622,148.185
C09907=1229.465,286.014,-65.000,-176.499,6.624,148.185
C09908=1229.461,286.262,-65.028,-176.497,6.626,148.184
C09909=1229.456,286.511,-65.056,-176.495,6.629,148.184
C09910=1229.451,286.759,-65.085,-176.492,6.631,148.184
C09911=1229.448,287.007,-65.114,-176.490,6.634,148.184
C09912=1229.443,287.256,-65.142,-176.487,6.636,148.184
C09913=1229.439,287.504,-65.170,-176.485,6.638,148.184
C09914=1229.435,287.752,-65.199,-176.483,6.640,148.184
C09915=1229.430,288.001,-65.228,-176.480,6.643,148.183
C09916=1229.426,288.249,-65.256,-176.478,6.645,148.183
C09917=1229.421,288.498,-65.285,-176.476,6.647,148.183
C09918=1229.417,288.746,-65.314,-176.473,6.649,148.183
C09919=1229.413,288.994,-65.342,-176.471,6.651,148.183
C09920=1229.408,289.269,-65.374,-176.468,6.654,148.183
C09921=1229.403,289.542,-65.406,-176.465,6.657,148.183
C09922=1229.398,289.816,-65.437,-176.463,6.659,148.183
C09923=1229.393,290.090,-65.469,-176.460,6.662,148.182
C09924=1229.389,290.339,-65.498,-176.458,6.664,148.182
C09925=1229.385,290.587,-65.526,-176.456,6.666,148.182
C09926=1229.380,290.835,-65.555,-176.453,6.668,148.182
C09927=1229.376,291.084,-65.584,-176.450,6.671,148.182
C09928=1229.372,291.332,-65.612,-176.448,6.674,148.182
C09929=1229.368,291.580,-65.642,-176.446,6.676,148.182
C09930=1229.363,291.829,-65.670,-176.444,6.678,148.182
C09931=1229.359,292.077,-65.700,-176.441,6.680,148.182
C09932=1229.354,292.325,-65.727,-176.439,6.683,148.182
C09933=1229.350,292.573,-65.757,-176.436,6.685,148.181
C09934=1229.346,292.822,-65.786,-176.434,6.687,148.181
C09935=1229.342,293.070,-65.815,-176.432,6.689,148.181
C09936=1229.337,293.318,-65.843,-176.429,6.692,148.181
C09937=1229.333,293.566,-65.872,-176.427,6.694,148.181
C09938=1229.329,293.815,-65.901,-176.425,6.697,148.181
C09939=1229.324,294.063,-65.930,-176.423,6.699,148.181
C09940=1229.319,294.312,-65.959,-176.419,6.701,148.180
C09941=1229.315,294.560,-65.988,-176.417,6.704,148.180
C09942=1229.312,294.808,-66.017,-176.415,6.706,148.180
C09943=1229.307,295.056,-66.046,-176.413,6.708,148.180
C09944=1229.302,295.304,-66.075,-176.410,6.711,148.180
C09945=1229.298,295.553,-66.104,-176.408,6.713,148.180
C09946=1229.294,295.802,-66.133,-176.406,6.715,148.180
C09947=1229.289,296.049,-66.162,-176.404,6.718,148.180
C09948=1229.285,296.297,-66.192,-176.401,6.720,148.180
C09949=1229.281,296.546,-66.220,-176.398,6.723,148.180
C09950=1229.277,296.794,-66.249,-176.396,6.725,148.180
C09951=1229.273,297.042,-66.279,-176.394,6.727,148.179
C09952=1229.268,297.291,-66.307,-176.392,6.730,148.179
C09953=1229.263,297.539,-66.337,-176.389,6.732,148.179
C09954=1229.259,297.787,-66.366,-176.387,6.734,148.179
C09955=1229.255,298.035,-66.396,-176.385,6.736,148.179
C09956=1229.251,298.284,-66.424,-176.382,6.739,148.179
C09957=1229.246,298.532,-66.453,-176.380,6.742,148.179
C09958=1229.242,298.780,-66.483,-176.377,6.744,148.179
C09959=1229.237,299.028,-66.512,-176.375,6.746,148.179
C09960=1229.233,299.277,-66.542,-176.373,6.749,148.179
C09961=1229.229,299.526,-66.570,-176.371,6.751,148.179
C09962=1229.225,299.774,-66.600,-176.368,6.753,148.179
C09963=1229.220,300.021,-66.629,-176.366,6.755,148.178
C09964=1229.216,300.269,-66.658,-176.363,6.758,148.178
C09965=1229.211,300.518,-66.688,-176.361,6.760,148.178
C09966=1229.207,300.766,-66.717,-176.359,6.763,148.178
C09967=1229.203,301.015,-66.747,-176.357,6.765,148.178
C09968=1229.199,301.263,-66.776,-176.354,6.768,148.178
C09969=1229.194,301.511,-66.805,-176.352,6.770,148.178
C09970=1229.190,301.759,-66.834,-176.350,6.772,148.178
C09971=1229.185,302.007,-66.864,-176.347,6.774,148.178
C09972=1229.181,302.256,-66.893,-176.345,6.777,148.178
C09973=1229.177,302.504,-66.922,-176.343,6.780,148.178
C09974=1229.173,302.752,-66.952,-176.341,6.782,148.178
C09975=1229.169,303.001,-66.981,-176.338,6.785,148.178
C09976=1229.165,303.249,-67.011,-176.336,6.787,148.178
C09977=1229.160,303.497,-67.040,-176.334,6.789,148.177
C09978=1229.156,303.745,-67.069,-176.332,6.792,148.177
C09979=1229.151,303.993,-67.099,-176.329,6.795,148.177
C09980=1229.147,304.241,-67.128,-176.327,6.797,148.177
C09981=1229.142,304.490,-67.158,-176.324,6.799,148.177
C09982=1229.138,304.738,-67.188,-176.322,6.801,148.177
C09983=1229.134,304.986,-67.217,-176.319,6.804,148.177
C09984=1229.130,305.235,-67.247,-176.317,6.806,148.177
C09985=1229.126,305.482,-67.277,-176.315,6.808,148.177
C09986=1229.122,305.730,-67.306,-176.313,6.811,148.177
C09987=1229.118,305.979,-67.336,-176.310,6.814,148.177
C09988=1229.113,306.227,-67.366,-176.308,6.816,148.177
C09989=1229.108,306.476,-67.395,-176.306,6.818,148.177
C09990=1229.104,306.724,-67.425,-176.304,6.821,148.177
C09991=1229.100,306.972,-67.454,-176.302,6.823,148.177
C09992=1229.096,307.219,-67.484,-176.299,6.826,148.177
C09993=1229.091,307.468,-67.514,-176.297,6.829,148.177
C09994=1229.086,307.716,-67.543,-176.295,6.831,148.177
C09995=1229.082,307.964,-67.573,-176.293,6.833,148.177
C09996=1229.078,308.212,-67.602,-176.290,6.835,148.176
//INST
///DATE 2021/06/25 14:26
///ATTR SC,RW,RJ
////FRAME ROBOT
///GROUP1 RB1
NOP
MOVL C00000 V=800.0 PL=0
MOVL C00001 V=800.0 PL=0
MOVL C00002 V=800.0 PL=0
MOVL C00003 V=800.0 PL=0
MOVL C00004 V=800.0 PL=0
MOVL C00005 V=800.0 PL=0
MOVL C00006 V=800.0 PL=0
MOVL C00007 V=800.0 PL=0
MOVL C00008 V=800.0 PL=0
MOVL C00009 V=800.0 PL=0
MOVL C00010 V=800.0 PL=0
MOVL C00011 V=800.0 PL=0
MOVL C00012 V=800.0 PL=0
MOVL C00013 V=800.0 PL=0
MOVL C00014 V=800.0 PL=0
MOVL C00015 V=800.0 PL=0
MOVL C00016 V=800.0 PL=0
MOVL C00017 V=800.0 PL=0
MOVL C00018 V=800.0 PL=0
MOVL C00019 V=800.0 PL=0
MOVL C00020 V=800.0 PL=0
MOVL C00021 V=800.0 PL=0
MOVL C00022 V=800.0 PL=0
MOVL C00023 V=800.0 PL=0
MOVL C00024 V=800.0 PL=0
MOVL C00025 V=800.0 PL=0
MOVL C00026 V=800.0 PL=0
MOVL C00027 V=800.0 PL=0
MOVL C00028 V=800.0 PL=0
MOVL C00029 V=800.0 PL=0
MOVL C00030 V=800.0 PL=0
MOVL C00031 V=800.0 PL=0
MOVL C00032 V=800.0 PL=0
MOVL C00033 V=800.0 PL=0
MOVL C00034 V=800.0 PL=0
MOVL C00035 V=800.0 PL=0
MOVL C00036 V=800.0 PL=0
MOVL C00037 V=800.0 PL=0
MOVL C00038 V=800.0 PL=0
MOVL C00039 V=800.0 PL=0
MOVL C00040 V=800.0 PL=0
MOVL C00041 V=800.0 PL=0
MOVL C00042 V=800.0 PL=0
MOVL C00043 V=800.0 PL=0
MOVL C00044 V=800.0 PL=0
MOVL C00045 V=800.0 PL=0
MOVL C00046 V=800.0 PL=0
MOVL C00047 V=800.0 PL=0
MOVL C00048 V=800.0 PL=0
MOVL C00049 V=800.0 PL=0
MOVL C00050 V=800.0 PL=0
MOVL C00051 V=800.0 PL=0
MOVL C00052 V=800.0 PL=0
MOVL C00053 V=800.0 PL=0
MOVL C00054 V=800.0 PL=0
MOVL C00055 V=800.0 PL=0
MOVL C00056 V=800.0 PL=0
MOVL C00057 V=800.0 PL=0
MOVL C00058 V=800.0 PL=0
MOVL C00059 V=800.0 PL=0
MOVL C00060 V=800.0 PL=0
MOVL C00061 V=800.0 PL=0
MOVL C00062 V=800.0 PL=0
MOVL C00063 V=800.0 PL=0
MOVL C00064 V=800.0 PL=0
MOVL C00065 V=800.0 PL=0
MOVL C00066 V=800.0 PL=0
MOVL C00067 V=800.0 PL=0
MOVL C00068 V=800.0 PL=0
MOVL C00069 V=800.0 PL=0
MOVL C00070 V=800.0 PL=0
MOVL C00071 V=800.0 PL=0
MOVL C00072 V=800.0 PL=0
MOVL C00073 V=800.0 PL=0
MOVL C00074 V=800.0 PL=0
MOVL C00075 V=800.0 PL=0
MOVL C00076 V=800.0 PL=0
MOVL C00077 V=800.0 PL=0
MOVL C00078 V=800.0 PL=0
MOVL C00079 V=800.0 PL=0
MOVL C00080 V=800.0 PL=0
MOVL C00081 V=800.0 PL=0
MOVL C00082 V=800.0 PL=0
MOVL C00083 V=800.0 PL=0
MOVL C00084 V=800.0 PL=0
MOVL C00085 V=800.0 PL=0
MOVL C00086 V=800.0 PL=0
MOVL C00087 V=800.0 PL=0
MOVL C00088 V=800.0 PL=0
MOVL C00089 V=800.0 PL=0
MOVL C00090 V=800.0 PL=0
MOVL C00091 V=800.0 PL=0
MOVL C00092 V=800.0 PL=0
MOVL C00093 V=800.0 PL=0
MOVL C00094 V=800.0 PL=0
MOVL C00095 V=800.0 PL=0
MOVL C00096 V=800.0 PL=0
MOVL C00097 V=800.0 PL=0
MOVL C00098 V=800.0 PL=0
MOVL C00099 V=800.0 PL=0
MOVL C00100 V=800.0 PL=0
MOVL C00101 V=800.0 PL=0
MOVL C00102 V=800.0 PL=0
MOVL C00103 V=800.0 PL=0
MOVL C00104 V=800.0 PL=0
MOVL C00105 V=800.0 PL=0
MOVL C00106 V=800.0 PL=0
MOVL C00107 V=800.0 PL=0
MOVL C00108 V=800.0 PL=0
MOVL C00109 V=800.0 PL=0
MOVL C00110 V=800.0 PL=0
MOVL C00111 V=800.0 PL=0
MOVL C00112 V=800.0 PL=0
MOVL C00113 V=800.0 PL=0
MOVL C00114 V=800.0 PL=0
MOVL C00115 V=800.0 PL=0
MOVL C00116 V=800.0 PL=0
MOVL C00117 V=800.0 PL=0
MOVL C00118 V=800.0 PL=0
MOVL C00119 V=800.0 PL=0
MOVL C00120 V=800.0 PL=0
MOVL C00121 V=800.0 PL=0
MOVL C00122 V=800.0 PL=0
MOVL C00123 V=800.0 PL=0
MOVL C00124 V=800.0 PL=0
MOVL C00125 V=800.0 PL=0
MOVL C00126 V=800.0 PL=0
MOVL C00127 V=800.0 PL=0
MOVL C00128 V=800.0 PL=0
MOVL C00129 V=800.0 PL=0
MOVL C00130 V=800.0 PL=0
MOVL C00131 V=800.0 PL=0
MOVL C00132 V=800.0 PL=0
MOVL C00133 V=800.0 PL=0
MOVL C00134 V=800.0 PL=0
MOVL C00135 V=800.0 PL=0
MOVL C00136 V=800.0 PL=0
MOVL C00137 V=800.0 PL=0
MOVL C00138 V=800.0 PL=0
MOVL C00139 V=800.0 PL=0
MOVL C00140 V=800.0 PL=0
MOVL C00141 V=800.0 PL=0
MOVL C00142 V=800.0 PL=0
MOVL C00143 V=800.0 PL=0
MOVL C00144 V=800.0 PL=0
MOVL C00145 V=800.0 PL=0
MOVL C00146 V=800.0 PL=0
MOVL C00147 V=800.0 PL=0
MOVL C00148 V=800.0 PL=0
MOVL C00149 V=800.0 PL=0
MOVL C00150 V=800.0 PL=0
MOVL C00151 V=800.0 PL=0
MOVL C00152 V=800.0 PL=0
MOVL C00153 V=800.0 PL=0
MOVL C00154 V=800.0 PL=0
MOVL C00155 V=800.0 PL=0
MOVL C00156 V=800.0 PL=0
MOVL C00157 V=800.0 PL=0
MOVL C00158 V=800.0 PL=0
MOVL C00159 V=800.0 PL=0
MOVL C00160 V=800.0 PL=0
MOVL C00161 V=800.0 PL=0
MOVL C00162 V=800.0 PL=0
MOVL C00163 V=800.0 PL=0
MOVL C00164 V=800.0 PL=0
MOVL C00165 V=800.0 PL=0
MOVL C00166 V=800.0 PL=0
MOVL C00167 V=800.0 PL=0
MOVL C00168 V=800.0 PL=0
MOVL C00169 V=800.0 PL=0
MOVL C00170 V=800.0 PL=0
MOVL C00171 V=800.0 PL=0
MOVL C00172 V=800.0 PL=0
MOVL C00173 V=800.0 PL=0
MOVL C00174 V=800.0 PL=0
MOVL C00175 V=800.0 PL=0
MOVL C00176 V=800.0 PL=0
MOVL C00177 V=800.0 PL=0
MOVL C00178 V=800.0 PL=0
MOVL C00179 V=800.0 PL=0
MOVL C00180 V=800.0 PL=0
MOVL C00181 V=800.0 PL=0
MOVL C00182 V=800.0 PL=0
MOVL C00183 V=800.0 PL=0
MOVL C00184 V=800.0 PL=0
MOVL C00185 V=800.0 PL=0
MOVL C00186 V=800.0 PL=0
MOVL C00187 V=800.0 PL=0
MOVL C00188 V=800.0 PL=0
MOVL C00189 V=800.0 PL=0
MOVL C00190 V=800.0 PL=0
MOVL C00191 V=800.0 PL=0
MOVL C00192 V=800.0 PL=0
MOVL C00193 V=800.0 PL=0
MOVL C00194 V=800.0 PL=0
MOVL C00195 V=800.0 PL=0
MOVL C00196 V=800.0 PL=0
MOVL C00197 V=800.0 PL=0
MOVL C00198 V=800.0 PL=0
MOVL C00199 V=800.0 PL=0
MOVL C00200 V=800.0 PL=0
MOVL C00201 V=800.0 PL=0
MOVL C00202 V=800.0 PL=0
MOVL C00203 V=800.0 PL=0
MOVL C00204 V=800.0 PL=0
MOVL C00205 V=800.0 PL=0
MOVL C00206 V=800.0 PL=0
MOVL C00207 V=800.0 PL=0
MOVL C00208 V=800.0 PL=0
MOVL C00209 V=800.0 PL=0
MOVL C00210 V=800.0 PL=0
MOVL C00211 V=800.0 PL=0
MOVL C00212 V=800.0 PL=0
MOVL C00213 V=800.0 PL=0
MOVL C00214 V=800.0 PL=0
MOVL C00215 V=800.0 PL=0
MOVL C00216 V=800.0 PL=0
MOVL C00217 V=800.0 PL=0
MOVL C00218 V=800.0 PL=0
MOVL C00219 V=800.0 PL=0
MOVL C00220 V=800.0 PL=0
MOVL C00221 V=800.0 PL=0
MOVL C00222 V=800.0 PL=0
MOVL C00223 V=800.0 PL=0
MOVL C00224 V=800.0 PL=0
MOVL C00225 V=800.0 PL=0
MOVL C00226 V=800.0 PL=0
MOVL C00227 V=800.0 PL=0
MOVL C00228 V=800.0 PL=0
MOVL C00229 V=800.0 PL=0
MOVL C00230 V=800.0 PL=0
MOVL C00231 V=800.0 PL=0
MOVL C00232 V=800.0 PL=0
MOVL C00233 V=800.0 PL=0
MOVL C00234 V=800.0 PL=0
MOVL C00235 V=800.0 PL=0
MOVL C00236 V=800.0 PL=0
MOVL C00237 V=800.0 PL=0
MOVL C00238 V=800.0 PL=0
MOVL C00239 V=800.0 PL=0
MOVL C00240 V=800.0 PL=0
MOVL C00241 V=800.0 PL=0
MOVL C00242 V=800.0 PL=0
MOVL C00243 V=800.0 PL=0
MOVL C00244 V=800.0 PL=0
MOVL C00245 V=800.0 PL=0
MOVL C00246 V=800.0 PL=0
MOVL C00247 V=800.0 PL=0
MOVL C00248 V=800.0 PL=0
MOVL C00249 V=800.0 PL=0
MOVL C00250 V=800.0 PL=0
MOVL C00251 V=800.0 PL=0
MOVL C00252 V=800.0 PL=0
MOVL C00253 V=800.0 PL=0
MOVL C00254 V=800.0 PL=0
MOVL C00255 V=800.0 PL=0
MOVL C00256 V=800.0 PL=0
MOVL C00257 V=800.0 PL=0
MOVL C00258 V=800.0 PL=0
MOVL C00259 V=800.0 PL=0
MOVL C00260 V=800.0 PL=0
MOVL C00261 V=800.0 PL=0
MOVL C00262 V=800.0 PL=0
MOVL C00263 V=800.0 PL=0
MOVL C00264 V=800.0 PL=0
MOVL C00265 V=800.0 PL=0
MOVL C00266 V=800.0 PL=0
MOVL C00267 V=800.0 PL=0
MOVL C00268 V=800.0 PL=0
MOVL C00269 V=800.0 PL=0
MOVL C00270 V=800.0 PL=0
MOVL C00271 V=800.0 PL=0
MOVL C00272 V=800.0 PL=0
MOVL C00273 V=800.0 PL=0
MOVL C00274 V=800.0 PL=0
MOVL C00275 V=800.0 PL=0
MOVL C00276 V=800.0 PL=0
MOVL C00277 V=800.0 PL=0
MOVL C00278 V=800.0 PL=0
MOVL C00279 V=800.0 PL=0
MOVL C00280 V=800.0 PL=0
MOVL C00281 V=800.0 PL=0
MOVL C00282 V=800.0 PL=0
MOVL C00283 V=800.0 PL=0
MOVL C00284 V=800.0 PL=0
MOVL C00285 V=800.0 PL=0
MOVL C00286 V=800.0 PL=0
MOVL C00287 V=800.0 PL=0
MOVL C00288 V=800.0 PL=0
MOVL C00289 V=800.0 PL=0
MOVL C00290 V=800.0 PL=0
MOVL C00291 V=800.0 PL=0
MOVL C00292 V=800.0 PL=0
MOVL C00293 V=800.0 PL=0
MOVL C00294 V=800.0 PL=0
MOVL C00295 V=800.0 PL=0
MOVL C00296 V=800.0 PL=0
MOVL C00297 V=800.0 PL=0
MOVL C00298 V=800.0 PL=0
MOVL C00299 V=800.0 PL=0
MOVL C00300 V=800.0 PL=0
MOVL C00301 V=800.0 PL=0
MOVL C00302 V=800.0 PL=0
MOVL C00303 V=800.0 PL=0
MOVL C00304 V=800.0 PL=0
MOVL C00305 V=800.0 PL=0
MOVL C00306 V=800.0 PL=0
MOVL C00307 V=800.0 PL=0
MOVL C00308 V=800.0 PL=0
MOVL C00309 V=800.0 PL=0
MOVL C00310 V=800.0 PL=0
MOVL C00311 V=800.0 PL=0
MOVL C00312 V=800.0 PL=0
MOVL C00313 V=800.0 PL=0
MOVL C00314 V=800.0 PL=0
MOVL C00315 V=800.0 PL=0
MOVL C00316 V=800.0 PL=0
MOVL C00317 V=800.0 PL=0
MOVL C00318 V=800.0 PL=0
MOVL C00319 V=800.0 PL=0
MOVL C00320 V=800.0 PL=0
MOVL C00321 V=800.0 PL=0
MOVL C00322 V=800.0 PL=0
MOVL C00323 V=800.0 PL=0
MOVL C00324 V=800.0 PL=0
MOVL C00325 V=800.0 PL=0
MOVL C00326 V=800.0 PL=0
MOVL C00327 V=800.0 PL=0
MOVL C00328 V=800.0 PL=0
MOVL C00329 V=800.0 PL=0
MOVL C00330 V=800.0 PL=0
MOVL C00331 V=800.0 PL=0
MOVL C00332 V=800.0 PL=0
MOVL C00333 V=800.0 PL=0
MOVL C00334 V=800.0 PL=0
MOVL C00335 V=800.0 PL=0
MOVL C00336 V=800.0 PL=0
MOVL C00337 V=800.0 PL=0
MOVL C00338 V=800.0 PL=0
MOVL C00339 V=800.0 PL=0
MOVL C00340 V=800.0 PL=0
MOVL C00341 V=800.0 PL=0
MOVL C00342 V=800.0 PL=0
MOVL C00343 V=800.0 PL=0
MOVL C00344 V=800.0 PL=0
MOVL C00345 V=800.0 PL=0
MOVL C00346 V=800.0 PL=0
MOVL C00347 V=800.0 PL=0
MOVL C00348 V=800.0 PL=0
MOVL C00349 V=800.0 PL=0
MOVL C00350 V=800.0 PL=0
MOVL C00351 V=800.0 PL=0
MOVL C00352 V=800.0 PL=0
MOVL C00353 V=800.0 PL=0
MOVL C00354 V=800.0 PL=0
MOVL C00355 V=800.0 PL=0
MOVL C00356 V=800.0 PL=0
MOVL C00357 V=800.0 PL=0
MOVL C00358 V=800.0 PL=0
MOVL C00359 V=800.0 PL=0
MOVL C00360 V=800.0 PL=0
MOVL C00361 V=800.0 PL=0
MOVL C00362 V=800.0 PL=0
MOVL C00363 V=800.0 PL=0
MOVL C00364 V=800.0 PL=0
MOVL C00365 V=800.0 PL=0
MOVL C00366 V=800.0 PL=0
MOVL C00367 V=800.0 PL=0
MOVL C00368 V=800.0 PL=0
MOVL C00369 V=800.0 PL=0
MOVL C00370 V=800.0 PL=0
MOVL C00371 V=800.0 PL=0
MOVL C00372 V=800.0 PL=0
MOVL C00373 V=800.0 PL=0
MOVL C00374 V=800.0 PL=0
MOVL C00375 V=800.0 PL=0
MOVL C00376 V=800.0 PL=0
MOVL C00377 V=800.0 PL=0
MOVL C00378 V=800.0 PL=0
MOVL C00379 V=800.0 PL=0
MOVL C00380 V=800.0 PL=0
MOVL C00381 V=800.0 PL=0
MOVL C00382 V=800.0 PL=0
MOVL C00383 V=800.0 PL=0
MOVL C00384 V=800.0 PL=0
MOVL C00385 V=800.0 PL=0
MOVL C00386 V=800.0 PL=0
MOVL C00387 V=800.0 PL=0
MOVL C00388 V=800.0 PL=0
MOVL C00389 V=800.0 PL=0
MOVL C00390 V=800.0 PL=0
MOVL C00391 V=800.0 PL=0
MOVL C00392 V=800.0 PL=0
MOVL C00393 V=800.0 PL=0
MOVL C00394 V=800.0 PL=0
MOVL C00395 V=800.0 PL=0
MOVL C00396 V=800.0 PL=0
MOVL C00397 V=800.0 PL=0
MOVL C00398 V=800.0 PL=0
MOVL C00399 V=800.0 PL=0
MOVL C00400 V=800.0 PL=0
MOVL C00401 V=800.0 PL=0
MOVL C00402 V=800.0 PL=0
MOVL C00403 V=800.0 PL=0
MOVL C00404 V=800.0 PL=0
MOVL C00405 V=800.0 PL=0
MOVL C00406 V=800.0 PL=0
MOVL C00407 V=800.0 PL=0
MOVL C00408 V=800.0 PL=0
MOVL C00409 V=800.0 PL=0
MOVL C00410 V=800.0 PL=0
MOVL C00411 V=800.0 PL=0
MOVL C00412 V=800.0 PL=0
MOVL C00413 V=800.0 PL=0
MOVL C00414 V=800.0 PL=0
MOVL C00415 V=800.0 PL=0
MOVL C00416 V=800.0 PL=0
MOVL C00417 V=800.0 PL=0
MOVL C00418 V=800.0 PL=0
MOVL C00419 V=800.0 PL=0
MOVL C00420 V=800.0 PL=0
MOVL C00421 V=800.0 PL=0
MOVL C00422 V=800.0 PL=0
MOVL C00423 V=800.0 PL=0
MOVL C00424 V=800.0 PL=0
MOVL C00425 V=800.0 PL=0
MOVL C00426 V=800.0 PL=0
MOVL C00427 V=800.0 PL=0
MOVL C00428 V=800.0 PL=0
MOVL C00429 V=800.0 PL=0
MOVL C00430 V=800.0 PL=0
MOVL C00431 V=800.0 PL=0
MOVL C00432 V=800.0 PL=0
MOVL C00433 V=800.0 PL=0
MOVL C00434 V=800.0 PL=0
MOVL C00435 V=800.0 PL=0
MOVL C00436 V=800.0 PL=0
MOVL C00437 V=800.0 PL=0
MOVL C00438 V=800.0 PL=0
MOVL C00439 V=800.0 PL=0
MOVL C00440 V=800.0 PL=0
MOVL C00441 V=800.0 PL=0
MOVL C00442 V=800.0 PL=0
MOVL C00443 V=800.0 PL=0
MOVL C00444 V=800.0 PL=0
MOVL C00445 V=800.0 PL=0
MOVL C00446 V=800.0 PL=0
MOVL C00447 V=800.0 PL=0
MOVL C00448 V=800.0 PL=0
MOVL C00449 V=800.0 PL=0
MOVL C00450 V=800.0 PL=0
MOVL C00451 V=800.0 PL=0
MOVL C00452 V=800.0 PL=0
MOVL C00453 V=800.0 PL=0
MOVL C00454 V=800.0 PL=0
MOVL C00455 V=800.0 PL=0
MOVL C00456 V=800.0 PL=0
MOVL C00457 V=800.0 PL=0
MOVL C00458 V=800.0 PL=0
MOVL C00459 V=800.0 PL=0
MOVL C00460 V=800.0 PL=0
MOVL C00461 V=800.0 PL=0
MOVL C00462 V=800.0 PL=0
MOVL C00463 V=800.0 PL=0
MOVL C00464 V=800.0 PL=0
MOVL C00465 V=800.0 PL=0
MOVL C00466 V=800.0 PL=0
MOVL C00467 V=800.0 PL=0
MOVL C00468 V=800.0 PL=0
MOVL C00469 V=800.0 PL=0
MOVL C00470 V=800.0 PL=0
MOVL C00471 V=800.0 PL=0
MOVL C00472 V=800.0 PL=0
MOVL C00473 V=800.0 PL=0
MOVL C00474 V=800.0 PL=0
MOVL C00475 V=800.0 PL=0
MOVL C00476 V=800.0 PL=0
MOVL C00477 V=800.0 PL=0
MOVL C00478 V=800.0 PL=0
MOVL C00479 V=800.0 PL=0
MOVL C00480 V=800.0 PL=0
MOVL C00481 V=800.0 PL=0
MOVL C00482 V=800.0 PL=0
MOVL C00483 V=800.0 PL=0
MOVL C00484 V=800.0 PL=0
MOVL C00485 V=800.0 PL=0
MOVL C00486 V=800.0 PL=0
MOVL C00487 V=800.0 PL=0
MOVL C00488 V=800.0 PL=0
MOVL C00489 V=800.0 PL=0
MOVL C00490 V=800.0 PL=0
MOVL C00491 V=800.0 PL=0
MOVL C00492 V=800.0 PL=0
MOVL C00493 V=800.0 PL=0
MOVL C00494 V=800.0 PL=0
MOVL C00495 V=800.0 PL=0
MOVL C00496 V=800.0 PL=0
MOVL C00497 V=800.0 PL=0
MOVL C00498 V=800.0 PL=0
MOVL C00499 V=800.0 PL=0
MOVL C00500 V=800.0 PL=0
MOVL C00501 V=800.0 PL=0
MOVL C00502 V=800.0 PL=0
MOVL C00503 V=800.0 PL=0
MOVL C00504 V=800.0 PL=0
MOVL C00505 V=800.0 PL=0
MOVL C00506 V=800.0 PL=0
MOVL C00507 V=800.0 PL=0
MOVL C00508 V=800.0 PL=0
MOVL C00509 V=800.0 PL=0
MOVL C00510 V=800.0 PL=0
MOVL C00511 V=800.0 PL=0
MOVL C00512 V=800.0 PL=0
MOVL C00513 V=800.0 PL=0
MOVL C00514 V=800.0 PL=0
MOVL C00515 V=800.0 PL=0
MOVL C00516 V=800.0 PL=0
MOVL C00517 V=800.0 PL=0
MOVL C00518 V=800.0 PL=0
MOVL C00519 V=800.0 PL=0
MOVL C00520 V=800.0 PL=0
MOVL C00521 V=800.0 PL=0
MOVL C00522 V=800.0 PL=0
MOVL C00523 V=800.0 PL=0
MOVL C00524 V=800.0 PL=0
MOVL C00525 V=800.0 PL=0
MOVL C00526 V=800.0 PL=0
MOVL C00527 V=800.0 PL=0
MOVL C00528 V=800.0 PL=0
MOVL C00529 V=800.0 PL=0
MOVL C00530 V=800.0 PL=0
MOVL C00531 V=800.0 PL=0
MOVL C00532 V=800.0 PL=0
MOVL C00533 V=800.0 PL=0
MOVL C00534 V=800.0 PL=0
MOVL C00535 V=800.0 PL=0
MOVL C00536 V=800.0 PL=0
MOVL C00537 V=800.0 PL=0
MOVL C00538 V=800.0 PL=0
MOVL C00539 V=800.0 PL=0
MOVL C00540 V=800.0 PL=0
MOVL C00541 V=800.0 PL=0
MOVL C00542 V=800.0 PL=0
MOVL C00543 V=800.0 PL=0
MOVL C00544 V=800.0 PL=0
MOVL C00545 V=800.0 PL=0
MOVL C00546 V=800.0 PL=0
MOVL C00547 V=800.0 PL=0
MOVL C00548 V=800.0 PL=0
MOVL C00549 V=800.0 PL=0
MOVL C00550 V=800.0 PL=0
MOVL C00551 V=800.0 PL=0
MOVL C00552 V=800.0 PL=0
MOVL C00553 V=800.0 PL=0
MOVL C00554 V=800.0 PL=0
MOVL C00555 V=800.0 PL=0
MOVL C00556 V=800.0 PL=0
MOVL C00557 V=800.0 PL=0
MOVL C00558 V=800.0 PL=0
MOVL C00559 V=800.0 PL=0
MOVL C00560 V=800.0 PL=0
MOVL C00561 V=800.0 PL=0
MOVL C00562 V=800.0 PL=0
MOVL C00563 V=800.0 PL=0
MOVL C00564 V=800.0 PL=0
MOVL C00565 V=800.0 PL=0
MOVL C00566 V=800.0 PL=0
MOVL C00567 V=800.0 PL=0
MOVL C00568 V=800.0 PL=0
MOVL C00569 V=800.0 PL=0
MOVL C00570 V=800.0 PL=0
MOVL C00571 V=800.0 PL=0
MOVL C00572 V=800.0 PL=0
MOVL C00573 V=800.0 PL=0
MOVL C00574 V=800.0 PL=0
MOVL C00575 V=800.0 PL=0
MOVL C00576 V=800.0 PL=0
MOVL C00577 V=800.0 PL=0
MOVL C00578 V=800.0 PL=0
MOVL C00579 V=800.0 PL=0
MOVL C00580 V=800.0 PL=0
MOVL C00581 V=800.0 PL=0
MOVL C00582 V=800.0 PL=0
MOVL C00583 V=800.0 PL=0
MOVL C00584 V=800.0 PL=0
MOVL C00585 V=800.0 PL=0
MOVL C00586 V=800.0 PL=0
MOVL C00587 V=800.0 PL=0
MOVL C00588 V=800.0 PL=0
MOVL C00589 V=800.0 PL=0
MOVL C00590 V=800.0 PL=0
MOVL C00591 V=800.0 PL=0
MOVL C00592 V=800.0 PL=0
MOVL C00593 V=800.0 PL=0
MOVL C00594 V=800.0 PL=0
MOVL C00595 V=800.0 PL=0
MOVL C00596 V=800.0 PL=0
MOVL C00597 V=800.0 PL=0
MOVL C00598 V=800.0 PL=0
MOVL C00599 V=800.0 PL=0
MOVL C00600 V=800.0 PL=0
MOVL C00601 V=800.0 PL=0
MOVL C00602 V=800.0 PL=0
MOVL C00603 V=800.0 PL=0
MOVL C00604 V=800.0 PL=0
MOVL C00605 V=800.0 PL=0
MOVL C00606 V=800.0 PL=0
MOVL C00607 V=800.0 PL=0
MOVL C00608 V=800.0 PL=0
MOVL C00609 V=800.0 PL=0
MOVL C00610 V=800.0 PL=0
MOVL C00611 V=800.0 PL=0
MOVL C00612 V=800.0 PL=0
MOVL C00613 V=800.0 PL=0
MOVL C00614 V=800.0 PL=0
MOVL C00615 V=800.0 PL=0
MOVL C00616 V=800.0 PL=0
MOVL C00617 V=800.0 PL=0
MOVL C00618 V=800.0 PL=0
MOVL C00619 V=800.0 PL=0
MOVL C00620 V=800.0 PL=0
MOVL C00621 V=800.0 PL=0
MOVL C00622 V=800.0 PL=0
MOVL C00623 V=800.0 PL=0
MOVL C00624 V=800.0 PL=0
MOVL C00625 V=800.0 PL=0
MOVL C00626 V=800.0 PL=0
MOVL C00627 V=800.0 PL=0
MOVL C00628 V=800.0 PL=0
MOVL C00629 V=800.0 PL=0
MOVL C00630 V=800.0 PL=0
MOVL C00631 V=800.0 PL=0
MOVL C00632 V=800.0 PL=0
MOVL C00633 V=800.0 PL=0
MOVL C00634 V=800.0 PL=0
MOVL C00635 V=800.0 PL=0
MOVL C00636 V=800.0 PL=0
MOVL C00637 V=800.0 PL=0
MOVL C00638 V=800.0 PL=0
MOVL C00639 V=800.0 PL=0
MOVL C00640 V=800.0 PL=0
MOVL C00641 V=800.0 PL=0
MOVL C00642 V=800.0 PL=0
MOVL C00643 V=800.0 PL=0
MOVL C00644 V=800.0 PL=0
MOVL C00645 V=800.0 PL=0
MOVL C00646 V=800.0 PL=0
MOVL C00647 V=800.0 PL=0
MOVL C00648 V=800.0 PL=0
MOVL C00649 V=800.0 PL=0
MOVL C00650 V=800.0 PL=0
MOVL C00651 V=800.0 PL=0
MOVL C00652 V=800.0 PL=0
MOVL C00653 V=800.0 PL=0
MOVL C00654 V=800.0 PL=0
MOVL C00655 V=800.0 PL=0
MOVL C00656 V=800.0 PL=0
MOVL C00657 V=800.0 PL=0
MOVL C00658 V=800.0 PL=0
MOVL C00659 V=800.0 PL=0
MOVL C00660 V=800.0 PL=0
MOVL C00661 V=800.0 PL=0
MOVL C00662 V=800.0 PL=0
MOVL C00663 V=800.0 PL=0
MOVL C00664 V=800.0 PL=0
MOVL C00665 V=800.0 PL=0
MOVL C00666 V=800.0 PL=0
MOVL C00667 V=800.0 PL=0
MOVL C00668 V=800.0 PL=0
MOVL C00669 V=800.0 PL=0
MOVL C00670 V=800.0 PL=0
MOVL C00671 V=800.0 PL=0
MOVL C00672 V=800.0 PL=0
MOVL C00673 V=800.0 PL=0
MOVL C00674 V=800.0 PL=0
MOVL C00675 V=800.0 PL=0
MOVL C00676 V=800.0 PL=0
MOVL C00677 V=800.0 PL=0
MOVL C00678 V=800.0 PL=0
MOVL C00679 V=800.0 PL=0
MOVL C00680 V=800.0 PL=0
MOVL C00681 V=800.0 PL=0
MOVL C00682 V=800.0 PL=0
MOVL C00683 V=800.0 PL=0
MOVL C00684 V=800.0 PL=0
MOVL C00685 V=800.0 PL=0
MOVL C00686 V=800.0 PL=0
MOVL C00687 V=800.0 PL=0
MOVL C00688 V=800.0 PL=0
MOVL C00689 V=800.0 PL=0
MOVL C00690 V=800.0 PL=0
MOVL C00691 V=800.0 PL=0
MOVL C00692 V=800.0 PL=0
MOVL C00693 V=800.0 PL=0
MOVL C00694 V=800.0 PL=0
MOVL C00695 V=800.0 PL=0
MOVL C00696 V=800.0 PL=0
MOVL C00697 V=800.0 PL=0
MOVL C00698 V=800.0 PL=0
MOVL C00699 V=800.0 PL=0
MOVL C00700 V=800.0 PL=0
MOVL C00701 V=800.0 PL=0
MOVL C00702 V=800.0 PL=0
MOVL C00703 V=800.0 PL=0
MOVL C00704 V=800.0 PL=0
MOVL C00705 V=800.0 PL=0
MOVL C00706 V=800.0 PL=0
MOVL C00707 V=800.0 PL=0
MOVL C00708 V=800.0 PL=0
MOVL C00709 V=800.0 PL=0
MOVL C00710 V=800.0 PL=0
MOVL C00711 V=800.0 PL=0
MOVL C00712 V=800.0 PL=0
MOVL C00713 V=800.0 PL=0
MOVL C00714 V=800.0 PL=0
MOVL C00715 V=800.0 PL=0
MOVL C00716 V=800.0 PL=0
MOVL C00717 V=800.0 PL=0
MOVL C00718 V=800.0 PL=0
MOVL C00719 V=800.0 PL=0
MOVL C00720 V=800.0 PL=0
MOVL C00721 V=800.0 PL=0
MOVL C00722 V=800.0 PL=0
MOVL C00723 V=800.0 PL=0
MOVL C00724 V=800.0 PL=0
MOVL C00725 V=800.0 PL=0
MOVL C00726 V=800.0 PL=0
MOVL C00727 V=800.0 PL=0
MOVL C00728 V=800.0 PL=0
MOVL C00729 V=800.0 PL=0
MOVL C00730 V=800.0 PL=0
MOVL C00731 V=800.0 PL=0
MOVL C00732 V=800.0 PL=0
MOVL C00733 V=800.0 PL=0
MOVL C00734 V=800.0 PL=0
MOVL C00735 V=800.0 PL=0
MOVL C00736 V=800.0 PL=0
MOVL C00737 V=800.0 PL=0
MOVL C00738 V=800.0 PL=0
MOVL C00739 V=800.0 PL=0
MOVL C00740 V=800.0 PL=0
MOVL C00741 V=800.0 PL=0
MOVL C00742 V=800.0 PL=0
MOVL C00743 V=800.0 PL=0
MOVL C00744 V=800.0 PL=0
MOVL C00745 V=800.0 PL=0
MOVL C00746 V=800.0 PL=0
MOVL C00747 V=800.0 PL=0
MOVL C00748 V=800.0 PL=0
MOVL C00749 V=800.0 PL=0
MOVL C00750 V=800.0 PL=0
MOVL C00751 V=800.0 PL=0
MOVL C00752 V=800.0 PL=0
MOVL C00753 V=800.0 PL=0
MOVL C00754 V=800.0 PL=0
MOVL C00755 V=800.0 PL=0
MOVL C00756 V=800.0 PL=0
MOVL C00757 V=800.0 PL=0
MOVL C00758 V=800.0 PL=0
MOVL C00759 V=800.0 PL=0
MOVL C00760 V=800.0 PL=0
MOVL C00761 V=800.0 PL=0
MOVL C00762 V=800.0 PL=0
MOVL C00763 V=800.0 PL=0
MOVL C00764 V=800.0 PL=0
MOVL C00765 V=800.0 PL=0
MOVL C00766 V=800.0 PL=0
MOVL C00767 V=800.0 PL=0
MOVL C00768 V=800.0 PL=0
MOVL C00769 V=800.0 PL=0
MOVL C00770 V=800.0 PL=0
MOVL C00771 V=800.0 PL=0
MOVL C00772 V=800.0 PL=0
MOVL C00773 V=800.0 PL=0
MOVL C00774 V=800.0 PL=0
MOVL C00775 V=800.0 PL=0
MOVL C00776 V=800.0 PL=0
MOVL C00777 V=800.0 PL=0
MOVL C00778 V=800.0 PL=0
MOVL C00779 V=800.0 PL=0
MOVL C00780 V=800.0 PL=0
MOVL C00781 V=800.0 PL=0
MOVL C00782 V=800.0 PL=0
MOVL C00783 V=800.0 PL=0
MOVL C00784 V=800.0 PL=0
MOVL C00785 V=800.0 PL=0
MOVL C00786 V=800.0 PL=0
MOVL C00787 V=800.0 PL=0
MOVL C00788 V=800.0 PL=0
MOVL C00789 V=800.0 PL=0
MOVL C00790 V=800.0 PL=0
MOVL C00791 V=800.0 PL=0
MOVL C00792 V=800.0 PL=0
MOVL C00793 V=800.0 PL=0
MOVL C00794 V=800.0 PL=0
MOVL C00795 V=800.0 PL=0
MOVL C00796 V=800.0 PL=0
MOVL C00797 V=800.0 PL=0
MOVL C00798 V=800.0 PL=0
MOVL C00799 V=800.0 PL=0
MOVL C00800 V=800.0 PL=0
MOVL C00801 V=800.0 PL=0
MOVL C00802 V=800.0 PL=0
MOVL C00803 V=800.0 PL=0
MOVL C00804 V=800.0 PL=0
MOVL C00805 V=800.0 PL=0
MOVL C00806 V=800.0 PL=0
MOVL C00807 V=800.0 PL=0
MOVL C00808 V=800.0 PL=0
MOVL C00809 V=800.0 PL=0
MOVL C00810 V=800.0 PL=0
MOVL C00811 V=800.0 PL=0
MOVL C00812 V=800.0 PL=0
MOVL C00813 V=800.0 PL=0
MOVL C00814 V=800.0 PL=0
MOVL C00815 V=800.0 PL=0
MOVL C00816 V=800.0 PL=0
MOVL C00817 V=800.0 PL=0
MOVL C00818 V=800.0 PL=0
MOVL C00819 V=800.0 PL=0
MOVL C00820 V=800.0 PL=0
MOVL C00821 V=800.0 PL=0
MOVL C00822 V=800.0 PL=0
MOVL C00823 V=800.0 PL=0
MOVL C00824 V=800.0 PL=0
MOVL C00825 V=800.0 PL=0
MOVL C00826 V=800.0 PL=0
MOVL C00827 V=800.0 PL=0
MOVL C00828 V=800.0 PL=0
MOVL C00829 V=800.0 PL=0
MOVL C00830 V=800.0 PL=0
MOVL C00831 V=800.0 PL=0
MOVL C00832 V=800.0 PL=0
MOVL C00833 V=800.0 PL=0
MOVL C00834 V=800.0 PL=0
MOVL C00835 V=800.0 PL=0
MOVL C00836 V=800.0 PL=0
MOVL C00837 V=800.0 PL=0
MOVL C00838 V=800.0 PL=0
MOVL C00839 V=800.0 PL=0
MOVL C00840 V=800.0 PL=0
MOVL C00841 V=800.0 PL=0
MOVL C00842 V=800.0 PL=0
MOVL C00843 V=800.0 PL=0
MOVL C00844 V=800.0 PL=0
MOVL C00845 V=800.0 PL=0
MOVL C00846 V=800.0 PL=0
MOVL C00847 V=800.0 PL=0
MOVL C00848 V=800.0 PL=0
MOVL C00849 V=800.0 PL=0
MOVL C00850 V=800.0 PL=0
MOVL C00851 V=800.0 PL=0
MOVL C00852 V=800.0 PL=0
MOVL C00853 V=800.0 PL=0
MOVL C00854 V=800.0 PL=0
MOVL C00855 V=800.0 PL=0
MOVL C00856 V=800.0 PL=0
MOVL C00857 V=800.0 PL=0
MOVL C00858 V=800.0 PL=0
MOVL C00859 V=800.0 PL=0
MOVL C00860 V=800.0 PL=0
MOVL C00861 V=800.0 PL=0
MOVL C00862 V=800.0 PL=0
MOVL C00863 V=800.0 PL=0
MOVL C00864 V=800.0 PL=0
MOVL C00865 V=800.0 PL=0
MOVL C00866 V=800.0 PL=0
MOVL C00867 V=800.0 PL=0
MOVL C00868 V=800.0 PL=0
MOVL C00869 V=800.0 PL=0
MOVL C00870 V=800.0 PL=0
MOVL C00871 V=800.0 PL=0
MOVL C00872 V=800.0 PL=0
MOVL C00873 V=800.0 PL=0
MOVL C00874 V=800.0 PL=0
MOVL C00875 V=800.0 PL=0
MOVL C00876 V=800.0 PL=0
MOVL C00877 V=800.0 PL=0
MOVL C00878 V=800.0 PL=0
MOVL C00879 V=800.0 PL=0
MOVL C00880 V=800.0 PL=0
MOVL C00881 V=800.0 PL=0
MOVL C00882 V=800.0 PL=0
MOVL C00883 V=800.0 PL=0
MOVL C00884 V=800.0 PL=0
MOVL C00885 V=800.0 PL=0
MOVL C00886 V=800.0 PL=0
MOVL C00887 V=800.0 PL=0
MOVL C00888 V=800.0 PL=0
MOVL C00889 V=800.0 PL=0
MOVL C00890 V=800.0 PL=0
MOVL C00891 V=800.0 PL=0
MOVL C00892 V=800.0 PL=0
MOVL C00893 V=800.0 PL=0
MOVL C00894 V=800.0 PL=0
MOVL C00895 V=800.0 PL=0
MOVL C00896 V=800.0 PL=0
MOVL C00897 V=800.0 PL=0
MOVL C00898 V=800.0 PL=0
MOVL C00899 V=800.0 PL=0
MOVL C00900 V=800.0 PL=0
MOVL C00901 V=800.0 PL=0
MOVL C00902 V=800.0 PL=0
MOVL C00903 V=800.0 PL=0
MOVL C00904 V=800.0 PL=0
MOVL C00905 V=800.0 PL=0
MOVL C00906 V=800.0 PL=0
MOVL C00907 V=800.0 PL=0
MOVL C00908 V=800.0 PL=0
MOVL C00909 V=800.0 PL=0
MOVL C00910 V=800.0 PL=0
MOVL C00911 V=800.0 PL=0
MOVL C00912 V=800.0 PL=0
MOVL C00913 V=800.0 PL=0
MOVL C00914 V=800.0 PL=0
MOVL C00915 V=800.0 PL=0
MOVL C00916 V=800.0 PL=0
MOVL C00917 V=800.0 PL=0
MOVL C00918 V=800.0 PL=0
MOVL C00919 V=800.0 PL=0
MOVL C00920 V=800.0 PL=0
MOVL C00921 V=800.0 PL=0
MOVL C00922 V=800.0 PL=0
MOVL C00923 V=800.0 PL=0
MOVL C00924 V=800.0 PL=0
MOVL C00925 V=800.0 PL=0
MOVL C00926 V=800.0 PL=0
MOVL C00927 V=800.0 PL=0
MOVL C00928 V=800.0 PL=0
MOVL C00929 V=800.0 PL=0
MOVL C00930 V=800.0 PL=0
MOVL C00931 V=800.0 PL=0
MOVL C00932 V=800.0 PL=0
MOVL C00933 V=800.0 PL=0
MOVL C00934 V=800.0 PL=0
MOVL C00935 V=800.0 PL=0
MOVL C00936 V=800.0 PL=0
MOVL C00937 V=800.0 PL=0
MOVL C00938 V=800.0 PL=0
MOVL C00939 V=800.0 PL=0
MOVL C00940 V=800.0 PL=0
MOVL C00941 V=800.0 PL=0
MOVL C00942 V=800.0 PL=0
MOVL C00943 V=800.0 PL=0
MOVL C00944 V=800.0 PL=0
MOVL C00945 V=800.0 PL=0
MOVL C00946 V=800.0 PL=0
MOVL C00947 V=800.0 PL=0
MOVL C00948 V=800.0 PL=0
MOVL C00949 V=800.0 PL=0
MOVL C00950 V=800.0 PL=0
MOVL C00951 V=800.0 PL=0
MOVL C00952 V=800.0 PL=0
MOVL C00953 V=800.0 PL=0
MOVL C00954 V=800.0 PL=0
MOVL C00955 V=800.0 PL=0
MOVL C00956 V=800.0 PL=0
MOVL C00957 V=800.0 PL=0
MOVL C00958 V=800.0 PL=0
MOVL C00959 V=800.0 PL=0
MOVL C00960 V=800.0 PL=0
MOVL C00961 V=800.0 PL=0
MOVL C00962 V=800.0 PL=0
MOVL C00963 V=800.0 PL=0
MOVL C00964 V=800.0 PL=0
MOVL C00965 V=800.0 PL=0
MOVL C00966 V=800.0 PL=0
MOVL C00967 V=800.0 PL=0
MOVL C00968 V=800.0 PL=0
MOVL C00969 V=800.0 PL=0
MOVL C00970 V=800.0 PL=0
MOVL C00971 V=800.0 PL=0
MOVL C00972 V=800.0 PL=0
MOVL C00973 V=800.0 PL=0
MOVL C00974 V=800.0 PL=0
MOVL C00975 V=800.0 PL=0
MOVL C00976 V=800.0 PL=0
MOVL C00977 V=800.0 PL=0
MOVL C00978 V=800.0 PL=0
MOVL C00979 V=800.0 PL=0
MOVL C00980 V=800.0 PL=0
MOVL C00981 V=800.0 PL=0
MOVL C00982 V=800.0 PL=0
MOVL C00983 V=800.0 PL=0
MOVL C00984 V=800.0 PL=0
MOVL C00985 V=800.0 PL=0
MOVL C00986 V=800.0 PL=0
MOVL C00987 V=800.0 PL=0
MOVL C00988 V=800.0 PL=0
MOVL C00989 V=800.0 PL=0
MOVL C00990 V=800.0 PL=0
MOVL C00991 V=800.0 PL=0
MOVL C00992 V=800.0 PL=0
MOVL C00993 V=800.0 PL=0
MOVL C00994 V=800.0 PL=0
MOVL C00995 V=800.0 PL=0
MOVL C00996 V=800.0 PL=0
MOVL C00997 V=800.0 PL=0
MOVL C00998 V=800.0 PL=0
MOVL C00999 V=800.0 PL=0
MOVL C01000 V=800.0 PL=0
MOVL C01001 V=800.0 PL=0
MOVL C01002 V=800.0 PL=0
MOVL C01003 V=800.0 PL=0
MOVL C01004 V=800.0 PL=0
MOVL C01005 V=800.0 PL=0
MOVL C01006 V=800.0 PL=0
MOVL C01007 V=800.0 PL=0
MOVL C01008 V=800.0 PL=0
MOVL C01009 V=800.0 PL=0
MOVL C01010 V=800.0 PL=0
MOVL C01011 V=800.0 PL=0
MOVL C01012 V=800.0 PL=0
MOVL C01013 V=800.0 PL=0
MOVL C01014 V=800.0 PL=0
MOVL C01015 V=800.0 PL=0
MOVL C01016 V=800.0 PL=0
MOVL C01017 V=800.0 PL=0
MOVL C01018 V=800.0 PL=0
MOVL C01019 V=800.0 PL=0
MOVL C01020 V=800.0 PL=0
MOVL C01021 V=800.0 PL=0
MOVL C01022 V=800.0 PL=0
MOVL C01023 V=800.0 PL=0
MOVL C01024 V=800.0 PL=0
MOVL C01025 V=800.0 PL=0
MOVL C01026 V=800.0 PL=0
MOVL C01027 V=800.0 PL=0
MOVL C01028 V=800.0 PL=0
MOVL C01029 V=800.0 PL=0
MOVL C01030 V=800.0 PL=0
MOVL C01031 V=800.0 PL=0
MOVL C01032 V=800.0 PL=0
MOVL C01033 V=800.0 PL=0
MOVL C01034 V=800.0 PL=0
MOVL C01035 V=800.0 PL=0
MOVL C01036 V=800.0 PL=0
MOVL C01037 V=800.0 PL=0
MOVL C01038 V=800.0 PL=0
MOVL C01039 V=800.0 PL=0
MOVL C01040 V=800.0 PL=0
MOVL C01041 V=800.0 PL=0
MOVL C01042 V=800.0 PL=0
MOVL C01043 V=800.0 PL=0
MOVL C01044 V=800.0 PL=0
MOVL C01045 V=800.0 PL=0
MOVL C01046 V=800.0 PL=0
MOVL C01047 V=800.0 PL=0
MOVL C01048 V=800.0 PL=0
MOVL C01049 V=800.0 PL=0
MOVL C01050 V=800.0 PL=0
MOVL C01051 V=800.0 PL=0
MOVL C01052 V=800.0 PL=0
MOVL C01053 V=800.0 PL=0
MOVL C01054 V=800.0 PL=0
MOVL C01055 V=800.0 PL=0
MOVL C01056 V=800.0 PL=0
MOVL C01057 V=800.0 PL=0
MOVL C01058 V=800.0 PL=0
MOVL C01059 V=800.0 PL=0
MOVL C01060 V=800.0 PL=0
MOVL C01061 V=800.0 PL=0
MOVL C01062 V=800.0 PL=0
MOVL C01063 V=800.0 PL=0
MOVL C01064 V=800.0 PL=0
MOVL C01065 V=800.0 PL=0
MOVL C01066 V=800.0 PL=0
MOVL C01067 V=800.0 PL=0
MOVL C01068 V=800.0 PL=0
MOVL C01069 V=800.0 PL=0
MOVL C01070 V=800.0 PL=0
MOVL C01071 V=800.0 PL=0
MOVL C01072 V=800.0 PL=0
MOVL C01073 V=800.0 PL=0
MOVL C01074 V=800.0 PL=0
MOVL C01075 V=800.0 PL=0
MOVL C01076 V=800.0 PL=0
MOVL C01077 V=800.0 PL=0
MOVL C01078 V=800.0 PL=0
MOVL C01079 V=800.0 PL=0
MOVL C01080 V=800.0 PL=0
MOVL C01081 V=800.0 PL=0
MOVL C01082 V=800.0 PL=0
MOVL C01083 V=800.0 PL=0
MOVL C01084 V=800.0 PL=0
MOVL C01085 V=800.0 PL=0
MOVL C01086 V=800.0 PL=0
MOVL C01087 V=800.0 PL=0
MOVL C01088 V=800.0 PL=0
MOVL C01089 V=800.0 PL=0
MOVL C01090 V=800.0 PL=0
MOVL C01091 V=800.0 PL=0
MOVL C01092 V=800.0 PL=0
MOVL C01093 V=800.0 PL=0
MOVL C01094 V=800.0 PL=0
MOVL C01095 V=800.0 PL=0
MOVL C01096 V=800.0 PL=0
MOVL C01097 V=800.0 PL=0
MOVL C01098 V=800.0 PL=0
MOVL C01099 V=800.0 PL=0
MOVL C01100 V=800.0 PL=0
MOVL C01101 V=800.0 PL=0
MOVL C01102 V=800.0 PL=0
MOVL C01103 V=800.0 PL=0
MOVL C01104 V=800.0 PL=0
MOVL C01105 V=800.0 PL=0
MOVL C01106 V=800.0 PL=0
MOVL C01107 V=800.0 PL=0
MOVL C01108 V=800.0 PL=0
MOVL C01109 V=800.0 PL=0
MOVL C01110 V=800.0 PL=0
MOVL C01111 V=800.0 PL=0
MOVL C01112 V=800.0 PL=0
MOVL C01113 V=800.0 PL=0
MOVL C01114 V=800.0 PL=0
MOVL C01115 V=800.0 PL=0
MOVL C01116 V=800.0 PL=0
MOVL C01117 V=800.0 PL=0
MOVL C01118 V=800.0 PL=0
MOVL C01119 V=800.0 PL=0
MOVL C01120 V=800.0 PL=0
MOVL C01121 V=800.0 PL=0
MOVL C01122 V=800.0 PL=0
MOVL C01123 V=800.0 PL=0
MOVL C01124 V=800.0 PL=0
MOVL C01125 V=800.0 PL=0
MOVL C01126 V=800.0 PL=0
MOVL C01127 V=800.0 PL=0
MOVL C01128 V=800.0 PL=0
MOVL C01129 V=800.0 PL=0
MOVL C01130 V=800.0 PL=0
MOVL C01131 V=800.0 PL=0
MOVL C01132 V=800.0 PL=0
MOVL C01133 V=800.0 PL=0
MOVL C01134 V=800.0 PL=0
MOVL C01135 V=800.0 PL=0
MOVL C01136 V=800.0 PL=0
MOVL C01137 V=800.0 PL=0
MOVL C01138 V=800.0 PL=0
MOVL C01139 V=800.0 PL=0
MOVL C01140 V=800.0 PL=0
MOVL C01141 V=800.0 PL=0
MOVL C01142 V=800.0 PL=0
MOVL C01143 V=800.0 PL=0
MOVL C01144 V=800.0 PL=0
MOVL C01145 V=800.0 PL=0
MOVL C01146 V=800.0 PL=0
MOVL C01147 V=800.0 PL=0
MOVL C01148 V=800.0 PL=0
MOVL C01149 V=800.0 PL=0
MOVL C01150 V=800.0 PL=0
MOVL C01151 V=800.0 PL=0
MOVL C01152 V=800.0 PL=0
MOVL C01153 V=800.0 PL=0
MOVL C01154 V=800.0 PL=0
MOVL C01155 V=800.0 PL=0
MOVL C01156 V=800.0 PL=0
MOVL C01157 V=800.0 PL=0
MOVL C01158 V=800.0 PL=0
MOVL C01159 V=800.0 PL=0
MOVL C01160 V=800.0 PL=0
MOVL C01161 V=800.0 PL=0
MOVL C01162 V=800.0 PL=0
MOVL C01163 V=800.0 PL=0
MOVL C01164 V=800.0 PL=0
MOVL C01165 V=800.0 PL=0
MOVL C01166 V=800.0 PL=0
MOVL C01167 V=800.0 PL=0
MOVL C01168 V=800.0 PL=0
MOVL C01169 V=800.0 PL=0
MOVL C01170 V=800.0 PL=0
MOVL C01171 V=800.0 PL=0
MOVL C01172 V=800.0 PL=0
MOVL C01173 V=800.0 PL=0
MOVL C01174 V=800.0 PL=0
MOVL C01175 V=800.0 PL=0
MOVL C01176 V=800.0 PL=0
MOVL C01177 V=800.0 PL=0
MOVL C01178 V=800.0 PL=0
MOVL C01179 V=800.0 PL=0
MOVL C01180 V=800.0 PL=0
MOVL C01181 V=800.0 PL=0
MOVL C01182 V=800.0 PL=0
MOVL C01183 V=800.0 PL=0
MOVL C01184 V=800.0 PL=0
MOVL C01185 V=800.0 PL=0
MOVL C01186 V=800.0 PL=0
MOVL C01187 V=800.0 PL=0
MOVL C01188 V=800.0 PL=0
MOVL C01189 V=800.0 PL=0
MOVL C01190 V=800.0 PL=0
MOVL C01191 V=800.0 PL=0
MOVL C01192 V=800.0 PL=0
MOVL C01193 V=800.0 PL=0
MOVL C01194 V=800.0 PL=0
MOVL C01195 V=800.0 PL=0
MOVL C01196 V=800.0 PL=0
MOVL C01197 V=800.0 PL=0
MOVL C01198 V=800.0 PL=0
MOVL C01199 V=800.0 PL=0
MOVL C01200 V=800.0 PL=0
MOVL C01201 V=800.0 PL=0
MOVL C01202 V=800.0 PL=0
MOVL C01203 V=800.0 PL=0
MOVL C01204 V=800.0 PL=0
MOVL C01205 V=800.0 PL=0
MOVL C01206 V=800.0 PL=0
MOVL C01207 V=800.0 PL=0
MOVL C01208 V=800.0 PL=0
MOVL C01209 V=800.0 PL=0
MOVL C01210 V=800.0 PL=0
MOVL C01211 V=800.0 PL=0
MOVL C01212 V=800.0 PL=0
MOVL C01213 V=800.0 PL=0
MOVL C01214 V=800.0 PL=0
MOVL C01215 V=800.0 PL=0
MOVL C01216 V=800.0 PL=0
MOVL C01217 V=800.0 PL=0
MOVL C01218 V=800.0 PL=0
MOVL C01219 V=800.0 PL=0
MOVL C01220 V=800.0 PL=0
MOVL C01221 V=800.0 PL=0
MOVL C01222 V=800.0 PL=0
MOVL C01223 V=800.0 PL=0
MOVL C01224 V=800.0 PL=0
MOVL C01225 V=800.0 PL=0
MOVL C01226 V=800.0 PL=0
MOVL C01227 V=800.0 PL=0
MOVL C01228 V=800.0 PL=0
MOVL C01229 V=800.0 PL=0
MOVL C01230 V=800.0 PL=0
MOVL C01231 V=800.0 PL=0
MOVL C01232 V=800.0 PL=0
MOVL C01233 V=800.0 PL=0
MOVL C01234 V=800.0 PL=0
MOVL C01235 V=800.0 PL=0
MOVL C01236 V=800.0 PL=0
MOVL C01237 V=800.0 PL=0
MOVL C01238 V=800.0 PL=0
MOVL C01239 V=800.0 PL=0
MOVL C01240 V=800.0 PL=0
MOVL C01241 V=800.0 PL=0
MOVL C01242 V=800.0 PL=0
MOVL C01243 V=800.0 PL=0
MOVL C01244 V=800.0 PL=0
MOVL C01245 V=800.0 PL=0
MOVL C01246 V=800.0 PL=0
MOVL C01247 V=800.0 PL=0
MOVL C01248 V=800.0 PL=0
MOVL C01249 V=800.0 PL=0
MOVL C01250 V=800.0 PL=0
MOVL C01251 V=800.0 PL=0
MOVL C01252 V=800.0 PL=0
MOVL C01253 V=800.0 PL=0
MOVL C01254 V=800.0 PL=0
MOVL C01255 V=800.0 PL=0
MOVL C01256 V=800.0 PL=0
MOVL C01257 V=800.0 PL=0
MOVL C01258 V=800.0 PL=0
MOVL C01259 V=800.0 PL=0
MOVL C01260 V=800.0 PL=0
MOVL C01261 V=800.0 PL=0
MOVL C01262 V=800.0 PL=0
MOVL C01263 V=800.0 PL=0
MOVL C01264 V=800.0 PL=0
MOVL C01265 V=800.0 PL=0
MOVL C01266 V=800.0 PL=0
MOVL C01267 V=800.0 PL=0
MOVL C01268 V=800.0 PL=0
MOVL C01269 V=800.0 PL=0
MOVL C01270 V=800.0 PL=0
MOVL C01271 V=800.0 PL=0
MOVL C01272 V=800.0 PL=0
MOVL C01273 V=800.0 PL=0
MOVL C01274 V=800.0 PL=0
MOVL C01275 V=800.0 PL=0
MOVL C01276 V=800.0 PL=0
MOVL C01277 V=800.0 PL=0
MOVL C01278 V=800.0 PL=0
MOVL C01279 V=800.0 PL=0
MOVL C01280 V=800.0 PL=0
MOVL C01281 V=800.0 PL=0
MOVL C01282 V=800.0 PL=0
MOVL C01283 V=800.0 PL=0
MOVL C01284 V=800.0 PL=0
MOVL C01285 V=800.0 PL=0
MOVL C01286 V=800.0 PL=0
MOVL C01287 V=800.0 PL=0
MOVL C01288 V=800.0 PL=0
MOVL C01289 V=800.0 PL=0
MOVL C01290 V=800.0 PL=0
MOVL C01291 V=800.0 PL=0
MOVL C01292 V=800.0 PL=0
MOVL C01293 V=800.0 PL=0
MOVL C01294 V=800.0 PL=0
MOVL C01295 V=800.0 PL=0
MOVL C01296 V=800.0 PL=0
MOVL C01297 V=800.0 PL=0
MOVL C01298 V=800.0 PL=0
MOVL C01299 V=800.0 PL=0
MOVL C01300 V=800.0 PL=0
MOVL C01301 V=800.0 PL=0
MOVL C01302 V=800.0 PL=0
MOVL C01303 V=800.0 PL=0
MOVL C01304 V=800.0 PL=0
MOVL C01305 V=800.0 PL=0
MOVL C01306 V=800.0 PL=0
MOVL C01307 V=800.0 PL=0
MOVL C01308 V=800.0 PL=0
MOVL C01309 V=800.0 PL=0
MOVL C01310 V=800.0 PL=0
MOVL C01311 V=800.0 PL=0
MOVL C01312 V=800.0 PL=0
MOVL C01313 V=800.0 PL=0
MOVL C01314 V=800.0 PL=0
MOVL C01315 V=800.0 PL=0
MOVL C01316 V=800.0 PL=0
MOVL C01317 V=800.0 PL=0
MOVL C01318 V=800.0 PL=0
MOVL C01319 V=800.0 PL=0
MOVL C01320 V=800.0 PL=0
MOVL C01321 V=800.0 PL=0
MOVL C01322 V=800.0 PL=0
MOVL C01323 V=800.0 PL=0
MOVL C01324 V=800.0 PL=0
MOVL C01325 V=800.0 PL=0
MOVL C01326 V=800.0 PL=0
MOVL C01327 V=800.0 PL=0
MOVL C01328 V=800.0 PL=0
MOVL C01329 V=800.0 PL=0
MOVL C01330 V=800.0 PL=0
MOVL C01331 V=800.0 PL=0
MOVL C01332 V=800.0 PL=0
MOVL C01333 V=800.0 PL=0
MOVL C01334 V=800.0 PL=0
MOVL C01335 V=800.0 PL=0
MOVL C01336 V=800.0 PL=0
MOVL C01337 V=800.0 PL=0
MOVL C01338 V=800.0 PL=0
MOVL C01339 V=800.0 PL=0
MOVL C01340 V=800.0 PL=0
MOVL C01341 V=800.0 PL=0
MOVL C01342 V=800.0 PL=0
MOVL C01343 V=800.0 PL=0
MOVL C01344 V=800.0 PL=0
MOVL C01345 V=800.0 PL=0
MOVL C01346 V=800.0 PL=0
MOVL C01347 V=800.0 PL=0
MOVL C01348 V=800.0 PL=0
MOVL C01349 V=800.0 PL=0
MOVL C01350 V=800.0 PL=0
MOVL C01351 V=800.0 PL=0
MOVL C01352 V=800.0 PL=0
MOVL C01353 V=800.0 PL=0
MOVL C01354 V=800.0 PL=0
MOVL C01355 V=800.0 PL=0
MOVL C01356 V=800.0 PL=0
MOVL C01357 V=800.0 PL=0
MOVL C01358 V=800.0 PL=0
MOVL C01359 V=800.0 PL=0
MOVL C01360 V=800.0 PL=0
MOVL C01361 V=800.0 PL=0
MOVL C01362 V=800.0 PL=0
MOVL C01363 V=800.0 PL=0
MOVL C01364 V=800.0 PL=0
MOVL C01365 V=800.0 PL=0
MOVL C01366 V=800.0 PL=0
MOVL C01367 V=800.0 PL=0
MOVL C01368 V=800.0 PL=0
MOVL C01369 V=800.0 PL=0
MOVL C01370 V=800.0 PL=0
MOVL C01371 V=800.0 PL=0
MOVL C01372 V=800.0 PL=0
MOVL C01373 V=800.0 PL=0
MOVL C01374 V=800.0 PL=0
MOVL C01375 V=800.0 PL=0
MOVL C01376 V=800.0 PL=0
MOVL C01377 V=800.0 PL=0
MOVL C01378 V=800.0 PL=0
MOVL C01379 V=800.0 PL=0
MOVL C01380 V=800.0 PL=0
MOVL C01381 V=800.0 PL=0
MOVL C01382 V=800.0 PL=0
MOVL C01383 V=800.0 PL=0
MOVL C01384 V=800.0 PL=0
MOVL C01385 V=800.0 PL=0
MOVL C01386 V=800.0 PL=0
MOVL C01387 V=800.0 PL=0
MOVL C01388 V=800.0 PL=0
MOVL C01389 V=800.0 PL=0
MOVL C01390 V=800.0 PL=0
MOVL C01391 V=800.0 PL=0
MOVL C01392 V=800.0 PL=0
MOVL C01393 V=800.0 PL=0
MOVL C01394 V=800.0 PL=0
MOVL C01395 V=800.0 PL=0
MOVL C01396 V=800.0 PL=0
MOVL C01397 V=800.0 PL=0
MOVL C01398 V=800.0 PL=0
MOVL C01399 V=800.0 PL=0
MOVL C01400 V=800.0 PL=0
MOVL C01401 V=800.0 PL=0
MOVL C01402 V=800.0 PL=0
MOVL C01403 V=800.0 PL=0
MOVL C01404 V=800.0 PL=0
MOVL C01405 V=800.0 PL=0
MOVL C01406 V=800.0 PL=0
MOVL C01407 V=800.0 PL=0
MOVL C01408 V=800.0 PL=0
MOVL C01409 V=800.0 PL=0
MOVL C01410 V=800.0 PL=0
MOVL C01411 V=800.0 PL=0
MOVL C01412 V=800.0 PL=0
MOVL C01413 V=800.0 PL=0
MOVL C01414 V=800.0 PL=0
MOVL C01415 V=800.0 PL=0
MOVL C01416 V=800.0 PL=0
MOVL C01417 V=800.0 PL=0
MOVL C01418 V=800.0 PL=0
MOVL C01419 V=800.0 PL=0
MOVL C01420 V=800.0 PL=0
MOVL C01421 V=800.0 PL=0
MOVL C01422 V=800.0 PL=0
MOVL C01423 V=800.0 PL=0
MOVL C01424 V=800.0 PL=0
MOVL C01425 V=800.0 PL=0
MOVL C01426 V=800.0 PL=0
MOVL C01427 V=800.0 PL=0
MOVL C01428 V=800.0 PL=0
MOVL C01429 V=800.0 PL=0
MOVL C01430 V=800.0 PL=0
MOVL C01431 V=800.0 PL=0
MOVL C01432 V=800.0 PL=0
MOVL C01433 V=800.0 PL=0
MOVL C01434 V=800.0 PL=0
MOVL C01435 V=800.0 PL=0
MOVL C01436 V=800.0 PL=0
MOVL C01437 V=800.0 PL=0
MOVL C01438 V=800.0 PL=0
MOVL C01439 V=800.0 PL=0
MOVL C01440 V=800.0 PL=0
MOVL C01441 V=800.0 PL=0
MOVL C01442 V=800.0 PL=0
MOVL C01443 V=800.0 PL=0
MOVL C01444 V=800.0 PL=0
MOVL C01445 V=800.0 PL=0
MOVL C01446 V=800.0 PL=0
MOVL C01447 V=800.0 PL=0
MOVL C01448 V=800.0 PL=0
MOVL C01449 V=800.0 PL=0
MOVL C01450 V=800.0 PL=0
MOVL C01451 V=800.0 PL=0
MOVL C01452 V=800.0 PL=0
MOVL C01453 V=800.0 PL=0
MOVL C01454 V=800.0 PL=0
MOVL C01455 V=800.0 PL=0
MOVL C01456 V=800.0 PL=0
MOVL C01457 V=800.0 PL=0
MOVL C01458 V=800.0 PL=0
MOVL C01459 V=800.0 PL=0
MOVL C01460 V=800.0 PL=0
MOVL C01461 V=800.0 PL=0
MOVL C01462 V=800.0 PL=0
MOVL C01463 V=800.0 PL=0
MOVL C01464 V=800.0 PL=0
MOVL C01465 V=800.0 PL=0
MOVL C01466 V=800.0 PL=0
MOVL C01467 V=800.0 PL=0
MOVL C01468 V=800.0 PL=0
MOVL C01469 V=800.0 PL=0
MOVL C01470 V=800.0 PL=0
MOVL C01471 V=800.0 PL=0
MOVL C01472 V=800.0 PL=0
MOVL C01473 V=800.0 PL=0
MOVL C01474 V=800.0 PL=0
MOVL C01475 V=800.0 PL=0
MOVL C01476 V=800.0 PL=0
MOVL C01477 V=800.0 PL=0
MOVL C01478 V=800.0 PL=0
MOVL C01479 V=800.0 PL=0
MOVL C01480 V=800.0 PL=0
MOVL C01481 V=800.0 PL=0
MOVL C01482 V=800.0 PL=0
MOVL C01483 V=800.0 PL=0
MOVL C01484 V=800.0 PL=0
MOVL C01485 V=800.0 PL=0
MOVL C01486 V=800.0 PL=0
MOVL C01487 V=800.0 PL=0
MOVL C01488 V=800.0 PL=0
MOVL C01489 V=800.0 PL=0
MOVL C01490 V=800.0 PL=0
MOVL C01491 V=800.0 PL=0
MOVL C01492 V=800.0 PL=0
MOVL C01493 V=800.0 PL=0
MOVL C01494 V=800.0 PL=0
MOVL C01495 V=800.0 PL=0
MOVL C01496 V=800.0 PL=0
MOVL C01497 V=800.0 PL=0
MOVL C01498 V=800.0 PL=0
MOVL C01499 V=800.0 PL=0
MOVL C01500 V=800.0 PL=0
MOVL C01501 V=800.0 PL=0
MOVL C01502 V=800.0 PL=0
MOVL C01503 V=800.0 PL=0
MOVL C01504 V=800.0 PL=0
MOVL C01505 V=800.0 PL=0
MOVL C01506 V=800.0 PL=0
MOVL C01507 V=800.0 PL=0
MOVL C01508 V=800.0 PL=0
MOVL C01509 V=800.0 PL=0
MOVL C01510 V=800.0 PL=0
MOVL C01511 V=800.0 PL=0
MOVL C01512 V=800.0 PL=0
MOVL C01513 V=800.0 PL=0
MOVL C01514 V=800.0 PL=0
MOVL C01515 V=800.0 PL=0
MOVL C01516 V=800.0 PL=0
MOVL C01517 V=800.0 PL=0
MOVL C01518 V=800.0 PL=0
MOVL C01519 V=800.0 PL=0
MOVL C01520 V=800.0 PL=0
MOVL C01521 V=800.0 PL=0
MOVL C01522 V=800.0 PL=0
MOVL C01523 V=800.0 PL=0
MOVL C01524 V=800.0 PL=0
MOVL C01525 V=800.0 PL=0
MOVL C01526 V=800.0 PL=0
MOVL C01527 V=800.0 PL=0
MOVL C01528 V=800.0 PL=0
MOVL C01529 V=800.0 PL=0
MOVL C01530 V=800.0 PL=0
MOVL C01531 V=800.0 PL=0
MOVL C01532 V=800.0 PL=0
MOVL C01533 V=800.0 PL=0
MOVL C01534 V=800.0 PL=0
MOVL C01535 V=800.0 PL=0
MOVL C01536 V=800.0 PL=0
MOVL C01537 V=800.0 PL=0
MOVL C01538 V=800.0 PL=0
MOVL C01539 V=800.0 PL=0
MOVL C01540 V=800.0 PL=0
MOVL C01541 V=800.0 PL=0
MOVL C01542 V=800.0 PL=0
MOVL C01543 V=800.0 PL=0
MOVL C01544 V=800.0 PL=0
MOVL C01545 V=800.0 PL=0
MOVL C01546 V=800.0 PL=0
MOVL C01547 V=800.0 PL=0
MOVL C01548 V=800.0 PL=0
MOVL C01549 V=800.0 PL=0
MOVL C01550 V=800.0 PL=0
MOVL C01551 V=800.0 PL=0
MOVL C01552 V=800.0 PL=0
MOVL C01553 V=800.0 PL=0
MOVL C01554 V=800.0 PL=0
MOVL C01555 V=800.0 PL=0
MOVL C01556 V=800.0 PL=0
MOVL C01557 V=800.0 PL=0
MOVL C01558 V=800.0 PL=0
MOVL C01559 V=800.0 PL=0
MOVL C01560 V=800.0 PL=0
MOVL C01561 V=800.0 PL=0
MOVL C01562 V=800.0 PL=0
MOVL C01563 V=800.0 PL=0
MOVL C01564 V=800.0 PL=0
MOVL C01565 V=800.0 PL=0
MOVL C01566 V=800.0 PL=0
MOVL C01567 V=800.0 PL=0
MOVL C01568 V=800.0 PL=0
MOVL C01569 V=800.0 PL=0
MOVL C01570 V=800.0 PL=0
MOVL C01571 V=800.0 PL=0
MOVL C01572 V=800.0 PL=0
MOVL C01573 V=800.0 PL=0
MOVL C01574 V=800.0 PL=0
MOVL C01575 V=800.0 PL=0
MOVL C01576 V=800.0 PL=0
MOVL C01577 V=800.0 PL=0
MOVL C01578 V=800.0 PL=0
MOVL C01579 V=800.0 PL=0
MOVL C01580 V=800.0 PL=0
MOVL C01581 V=800.0 PL=0
MOVL C01582 V=800.0 PL=0
MOVL C01583 V=800.0 PL=0
MOVL C01584 V=800.0 PL=0
MOVL C01585 V=800.0 PL=0
MOVL C01586 V=800.0 PL=0
MOVL C01587 V=800.0 PL=0
MOVL C01588 V=800.0 PL=0
MOVL C01589 V=800.0 PL=0
MOVL C01590 V=800.0 PL=0
MOVL C01591 V=800.0 PL=0
MOVL C01592 V=800.0 PL=0
MOVL C01593 V=800.0 PL=0
MOVL C01594 V=800.0 PL=0
MOVL C01595 V=800.0 PL=0
MOVL C01596 V=800.0 PL=0
MOVL C01597 V=800.0 PL=0
MOVL C01598 V=800.0 PL=0
MOVL C01599 V=800.0 PL=0
MOVL C01600 V=800.0 PL=0
MOVL C01601 V=800.0 PL=0
MOVL C01602 V=800.0 PL=0
MOVL C01603 V=800.0 PL=0
MOVL C01604 V=800.0 PL=0
MOVL C01605 V=800.0 PL=0
MOVL C01606 V=800.0 PL=0
MOVL C01607 V=800.0 PL=0
MOVL C01608 V=800.0 PL=0
MOVL C01609 V=800.0 PL=0
MOVL C01610 V=800.0 PL=0
MOVL C01611 V=800.0 PL=0
MOVL C01612 V=800.0 PL=0
MOVL C01613 V=800.0 PL=0
MOVL C01614 V=800.0 PL=0
MOVL C01615 V=800.0 PL=0
MOVL C01616 V=800.0 PL=0
MOVL C01617 V=800.0 PL=0
MOVL C01618 V=800.0 PL=0
MOVL C01619 V=800.0 PL=0
MOVL C01620 V=800.0 PL=0
MOVL C01621 V=800.0 PL=0
MOVL C01622 V=800.0 PL=0
MOVL C01623 V=800.0 PL=0
MOVL C01624 V=800.0 PL=0
MOVL C01625 V=800.0 PL=0
MOVL C01626 V=800.0 PL=0
MOVL C01627 V=800.0 PL=0
MOVL C01628 V=800.0 PL=0
MOVL C01629 V=800.0 PL=0
MOVL C01630 V=800.0 PL=0
MOVL C01631 V=800.0 PL=0
MOVL C01632 V=800.0 PL=0
MOVL C01633 V=800.0 PL=0
MOVL C01634 V=800.0 PL=0
MOVL C01635 V=800.0 PL=0
MOVL C01636 V=800.0 PL=0
MOVL C01637 V=800.0 PL=0
MOVL C01638 V=800.0 PL=0
MOVL C01639 V=800.0 PL=0
MOVL C01640 V=800.0 PL=0
MOVL C01641 V=800.0 PL=0
MOVL C01642 V=800.0 PL=0
MOVL C01643 V=800.0 PL=0
MOVL C01644 V=800.0 PL=0
MOVL C01645 V=800.0 PL=0
MOVL C01646 V=800.0 PL=0
MOVL C01647 V=800.0 PL=0
MOVL C01648 V=800.0 PL=0
MOVL C01649 V=800.0 PL=0
MOVL C01650 V=800.0 PL=0
MOVL C01651 V=800.0 PL=0
MOVL C01652 V=800.0 PL=0
MOVL C01653 V=800.0 PL=0
MOVL C01654 V=800.0 PL=0
MOVL C01655 V=800.0 PL=0
MOVL C01656 V=800.0 PL=0
MOVL C01657 V=800.0 PL=0
MOVL C01658 V=800.0 PL=0
MOVL C01659 V=800.0 PL=0
MOVL C01660 V=800.0 PL=0
MOVL C01661 V=800.0 PL=0
MOVL C01662 V=800.0 PL=0
MOVL C01663 V=800.0 PL=0
MOVL C01664 V=800.0 PL=0
MOVL C01665 V=800.0 PL=0
MOVL C01666 V=800.0 PL=0
MOVL C01667 V=800.0 PL=0
MOVL C01668 V=800.0 PL=0
MOVL C01669 V=800.0 PL=0
MOVL C01670 V=800.0 PL=0
MOVL C01671 V=800.0 PL=0
MOVL C01672 V=800.0 PL=0
MOVL C01673 V=800.0 PL=0
MOVL C01674 V=800.0 PL=0
MOVL C01675 V=800.0 PL=0
MOVL C01676 V=800.0 PL=0
MOVL C01677 V=800.0 PL=0
MOVL C01678 V=800.0 PL=0
MOVL C01679 V=800.0 PL=0
MOVL C01680 V=800.0 PL=0
MOVL C01681 V=800.0 PL=0
MOVL C01682 V=800.0 PL=0
MOVL C01683 V=800.0 PL=0
MOVL C01684 V=800.0 PL=0
MOVL C01685 V=800.0 PL=0
MOVL C01686 V=800.0 PL=0
MOVL C01687 V=800.0 PL=0
MOVL C01688 V=800.0 PL=0
MOVL C01689 V=800.0 PL=0
MOVL C01690 V=800.0 PL=0
MOVL C01691 V=800.0 PL=0
MOVL C01692 V=800.0 PL=0
MOVL C01693 V=800.0 PL=0
MOVL C01694 V=800.0 PL=0
MOVL C01695 V=800.0 PL=0
MOVL C01696 V=800.0 PL=0
MOVL C01697 V=800.0 PL=0
MOVL C01698 V=800.0 PL=0
MOVL C01699 V=800.0 PL=0
MOVL C01700 V=800.0 PL=0
MOVL C01701 V=800.0 PL=0
MOVL C01702 V=800.0 PL=0
MOVL C01703 V=800.0 PL=0
MOVL C01704 V=800.0 PL=0
MOVL C01705 V=800.0 PL=0
MOVL C01706 V=800.0 PL=0
MOVL C01707 V=800.0 PL=0
MOVL C01708 V=800.0 PL=0
MOVL C01709 V=800.0 PL=0
MOVL C01710 V=800.0 PL=0
MOVL C01711 V=800.0 PL=0
MOVL C01712 V=800.0 PL=0
MOVL C01713 V=800.0 PL=0
MOVL C01714 V=800.0 PL=0
MOVL C01715 V=800.0 PL=0
MOVL C01716 V=800.0 PL=0
MOVL C01717 V=800.0 PL=0
MOVL C01718 V=800.0 PL=0
MOVL C01719 V=800.0 PL=0
MOVL C01720 V=800.0 PL=0
MOVL C01721 V=800.0 PL=0
MOVL C01722 V=800.0 PL=0
MOVL C01723 V=800.0 PL=0
MOVL C01724 V=800.0 PL=0
MOVL C01725 V=800.0 PL=0
MOVL C01726 V=800.0 PL=0
MOVL C01727 V=800.0 PL=0
MOVL C01728 V=800.0 PL=0
MOVL C01729 V=800.0 PL=0
MOVL C01730 V=800.0 PL=0
MOVL C01731 V=800.0 PL=0
MOVL C01732 V=800.0 PL=0
MOVL C01733 V=800.0 PL=0
MOVL C01734 V=800.0 PL=0
MOVL C01735 V=800.0 PL=0
MOVL C01736 V=800.0 PL=0
MOVL C01737 V=800.0 PL=0
MOVL C01738 V=800.0 PL=0
MOVL C01739 V=800.0 PL=0
MOVL C01740 V=800.0 PL=0
MOVL C01741 V=800.0 PL=0
MOVL C01742 V=800.0 PL=0
MOVL C01743 V=800.0 PL=0
MOVL C01744 V=800.0 PL=0
MOVL C01745 V=800.0 PL=0
MOVL C01746 V=800.0 PL=0
MOVL C01747 V=800.0 PL=0
MOVL C01748 V=800.0 PL=0
MOVL C01749 V=800.0 PL=0
MOVL C01750 V=800.0 PL=0
MOVL C01751 V=800.0 PL=0
MOVL C01752 V=800.0 PL=0
MOVL C01753 V=800.0 PL=0
MOVL C01754 V=800.0 PL=0
MOVL C01755 V=800.0 PL=0
MOVL C01756 V=800.0 PL=0
MOVL C01757 V=800.0 PL=0
MOVL C01758 V=800.0 PL=0
MOVL C01759 V=800.0 PL=0
MOVL C01760 V=800.0 PL=0
MOVL C01761 V=800.0 PL=0
MOVL C01762 V=800.0 PL=0
MOVL C01763 V=800.0 PL=0
MOVL C01764 V=800.0 PL=0
MOVL C01765 V=800.0 PL=0
MOVL C01766 V=800.0 PL=0
MOVL C01767 V=800.0 PL=0
MOVL C01768 V=800.0 PL=0
MOVL C01769 V=800.0 PL=0
MOVL C01770 V=800.0 PL=0
MOVL C01771 V=800.0 PL=0
MOVL C01772 V=800.0 PL=0
MOVL C01773 V=800.0 PL=0
MOVL C01774 V=800.0 PL=0
MOVL C01775 V=800.0 PL=0
MOVL C01776 V=800.0 PL=0
MOVL C01777 V=800.0 PL=0
MOVL C01778 V=800.0 PL=0
MOVL C01779 V=800.0 PL=0
MOVL C01780 V=800.0 PL=0
MOVL C01781 V=800.0 PL=0
MOVL C01782 V=800.0 PL=0
MOVL C01783 V=800.0 PL=0
MOVL C01784 V=800.0 PL=0
MOVL C01785 V=800.0 PL=0
MOVL C01786 V=800.0 PL=0
MOVL C01787 V=800.0 PL=0
MOVL C01788 V=800.0 PL=0
MOVL C01789 V=800.0 PL=0
MOVL C01790 V=800.0 PL=0
MOVL C01791 V=800.0 PL=0
MOVL C01792 V=800.0 PL=0
MOVL C01793 V=800.0 PL=0
MOVL C01794 V=800.0 PL=0
MOVL C01795 V=800.0 PL=0
MOVL C01796 V=800.0 PL=0
MOVL C01797 V=800.0 PL=0
MOVL C01798 V=800.0 PL=0
MOVL C01799 V=800.0 PL=0
MOVL C01800 V=800.0 PL=0
MOVL C01801 V=800.0 PL=0
MOVL C01802 V=800.0 PL=0
MOVL C01803 V=800.0 PL=0
MOVL C01804 V=800.0 PL=0
MOVL C01805 V=800.0 PL=0
MOVL C01806 V=800.0 PL=0
MOVL C01807 V=800.0 PL=0
MOVL C01808 V=800.0 PL=0
MOVL C01809 V=800.0 PL=0
MOVL C01810 V=800.0 PL=0
MOVL C01811 V=800.0 PL=0
MOVL C01812 V=800.0 PL=0
MOVL C01813 V=800.0 PL=0
MOVL C01814 V=800.0 PL=0
MOVL C01815 V=800.0 PL=0
MOVL C01816 V=800.0 PL=0
MOVL C01817 V=800.0 PL=0
MOVL C01818 V=800.0 PL=0
MOVL C01819 V=800.0 PL=0
MOVL C01820 V=800.0 PL=0
MOVL C01821 V=800.0 PL=0
MOVL C01822 V=800.0 PL=0
MOVL C01823 V=800.0 PL=0
MOVL C01824 V=800.0 PL=0
MOVL C01825 V=800.0 PL=0
MOVL C01826 V=800.0 PL=0
MOVL C01827 V=800.0 PL=0
MOVL C01828 V=800.0 PL=0
MOVL C01829 V=800.0 PL=0
MOVL C01830 V=800.0 PL=0
MOVL C01831 V=800.0 PL=0
MOVL C01832 V=800.0 PL=0
MOVL C01833 V=800.0 PL=0
MOVL C01834 V=800.0 PL=0
MOVL C01835 V=800.0 PL=0
MOVL C01836 V=800.0 PL=0
MOVL C01837 V=800.0 PL=0
MOVL C01838 V=800.0 PL=0
MOVL C01839 V=800.0 PL=0
MOVL C01840 V=800.0 PL=0
MOVL C01841 V=800.0 PL=0
MOVL C01842 V=800.0 PL=0
MOVL C01843 V=800.0 PL=0
MOVL C01844 V=800.0 PL=0
MOVL C01845 V=800.0 PL=0
MOVL C01846 V=800.0 PL=0
MOVL C01847 V=800.0 PL=0
MOVL C01848 V=800.0 PL=0
MOVL C01849 V=800.0 PL=0
MOVL C01850 V=800.0 PL=0
MOVL C01851 V=800.0 PL=0
MOVL C01852 V=800.0 PL=0
MOVL C01853 V=800.0 PL=0
MOVL C01854 V=800.0 PL=0
MOVL C01855 V=800.0 PL=0
MOVL C01856 V=800.0 PL=0
MOVL C01857 V=800.0 PL=0
MOVL C01858 V=800.0 PL=0
MOVL C01859 V=800.0 PL=0
MOVL C01860 V=800.0 PL=0
MOVL C01861 V=800.0 PL=0
MOVL C01862 V=800.0 PL=0
MOVL C01863 V=800.0 PL=0
MOVL C01864 V=800.0 PL=0
MOVL C01865 V=800.0 PL=0
MOVL C01866 V=800.0 PL=0
MOVL C01867 V=800.0 PL=0
MOVL C01868 V=800.0 PL=0
MOVL C01869 V=800.0 PL=0
MOVL C01870 V=800.0 PL=0
MOVL C01871 V=800.0 PL=0
MOVL C01872 V=800.0 PL=0
MOVL C01873 V=800.0 PL=0
MOVL C01874 V=800.0 PL=0
MOVL C01875 V=800.0 PL=0
MOVL C01876 V=800.0 PL=0
MOVL C01877 V=800.0 PL=0
MOVL C01878 V=800.0 PL=0
MOVL C01879 V=800.0 PL=0
MOVL C01880 V=800.0 PL=0
MOVL C01881 V=800.0 PL=0
MOVL C01882 V=800.0 PL=0
MOVL C01883 V=800.0 PL=0
MOVL C01884 V=800.0 PL=0
MOVL C01885 V=800.0 PL=0
MOVL C01886 V=800.0 PL=0
MOVL C01887 V=800.0 PL=0
MOVL C01888 V=800.0 PL=0
MOVL C01889 V=800.0 PL=0
MOVL C01890 V=800.0 PL=0
MOVL C01891 V=800.0 PL=0
MOVL C01892 V=800.0 PL=0
MOVL C01893 V=800.0 PL=0
MOVL C01894 V=800.0 PL=0
MOVL C01895 V=800.0 PL=0
MOVL C01896 V=800.0 PL=0
MOVL C01897 V=800.0 PL=0
MOVL C01898 V=800.0 PL=0
MOVL C01899 V=800.0 PL=0
MOVL C01900 V=800.0 PL=0
MOVL C01901 V=800.0 PL=0
MOVL C01902 V=800.0 PL=0
MOVL C01903 V=800.0 PL=0
MOVL C01904 V=800.0 PL=0
MOVL C01905 V=800.0 PL=0
MOVL C01906 V=800.0 PL=0
MOVL C01907 V=800.0 PL=0
MOVL C01908 V=800.0 PL=0
MOVL C01909 V=800.0 PL=0
MOVL C01910 V=800.0 PL=0
MOVL C01911 V=800.0 PL=0
MOVL C01912 V=800.0 PL=0
MOVL C01913 V=800.0 PL=0
MOVL C01914 V=800.0 PL=0
MOVL C01915 V=800.0 PL=0
MOVL C01916 V=800.0 PL=0
MOVL C01917 V=800.0 PL=0
MOVL C01918 V=800.0 PL=0
MOVL C01919 V=800.0 PL=0
MOVL C01920 V=800.0 PL=0
MOVL C01921 V=800.0 PL=0
MOVL C01922 V=800.0 PL=0
MOVL C01923 V=800.0 PL=0
MOVL C01924 V=800.0 PL=0
MOVL C01925 V=800.0 PL=0
MOVL C01926 V=800.0 PL=0
MOVL C01927 V=800.0 PL=0
MOVL C01928 V=800.0 PL=0
MOVL C01929 V=800.0 PL=0
MOVL C01930 V=800.0 PL=0
MOVL C01931 V=800.0 PL=0
MOVL C01932 V=800.0 PL=0
MOVL C01933 V=800.0 PL=0
MOVL C01934 V=800.0 PL=0
MOVL C01935 V=800.0 PL=0
MOVL C01936 V=800.0 PL=0
MOVL C01937 V=800.0 PL=0
MOVL C01938 V=800.0 PL=0
MOVL C01939 V=800.0 PL=0
MOVL C01940 V=800.0 PL=0
MOVL C01941 V=800.0 PL=0
MOVL C01942 V=800.0 PL=0
MOVL C01943 V=800.0 PL=0
MOVL C01944 V=800.0 PL=0
MOVL C01945 V=800.0 PL=0
MOVL C01946 V=800.0 PL=0
MOVL C01947 V=800.0 PL=0
MOVL C01948 V=800.0 PL=0
MOVL C01949 V=800.0 PL=0
MOVL C01950 V=800.0 PL=0
MOVL C01951 V=800.0 PL=0
MOVL C01952 V=800.0 PL=0
MOVL C01953 V=800.0 PL=0
MOVL C01954 V=800.0 PL=0
MOVL C01955 V=800.0 PL=0
MOVL C01956 V=800.0 PL=0
MOVL C01957 V=800.0 PL=0
MOVL C01958 V=800.0 PL=0
MOVL C01959 V=800.0 PL=0
MOVL C01960 V=800.0 PL=0
MOVL C01961 V=800.0 PL=0
MOVL C01962 V=800.0 PL=0
MOVL C01963 V=800.0 PL=0
MOVL C01964 V=800.0 PL=0
MOVL C01965 V=800.0 PL=0
MOVL C01966 V=800.0 PL=0
MOVL C01967 V=800.0 PL=0
MOVL C01968 V=800.0 PL=0
MOVL C01969 V=800.0 PL=0
MOVL C01970 V=800.0 PL=0
MOVL C01971 V=800.0 PL=0
MOVL C01972 V=800.0 PL=0
MOVL C01973 V=800.0 PL=0
MOVL C01974 V=800.0 PL=0
MOVL C01975 V=800.0 PL=0
MOVL C01976 V=800.0 PL=0
MOVL C01977 V=800.0 PL=0
MOVL C01978 V=800.0 PL=0
MOVL C01979 V=800.0 PL=0
MOVL C01980 V=800.0 PL=0
MOVL C01981 V=800.0 PL=0
MOVL C01982 V=800.0 PL=0
MOVL C01983 V=800.0 PL=0
MOVL C01984 V=800.0 PL=0
MOVL C01985 V=800.0 PL=0
MOVL C01986 V=800.0 PL=0
MOVL C01987 V=800.0 PL=0
MOVL C01988 V=800.0 PL=0
MOVL C01989 V=800.0 PL=0
MOVL C01990 V=800.0 PL=0
MOVL C01991 V=800.0 PL=0
MOVL C01992 V=800.0 PL=0
MOVL C01993 V=800.0 PL=0
MOVL C01994 V=800.0 PL=0
MOVL C01995 V=800.0 PL=0
MOVL C01996 V=800.0 PL=0
MOVL C01997 V=800.0 PL=0
MOVL C01998 V=800.0 PL=0
MOVL C01999 V=800.0 PL=0
MOVL C02000 V=800.0 PL=0
MOVL C02001 V=800.0 PL=0
MOVL C02002 V=800.0 PL=0
MOVL C02003 V=800.0 PL=0
MOVL C02004 V=800.0 PL=0
MOVL C02005 V=800.0 PL=0
MOVL C02006 V=800.0 PL=0
MOVL C02007 V=800.0 PL=0
MOVL C02008 V=800.0 PL=0
MOVL C02009 V=800.0 PL=0
MOVL C02010 V=800.0 PL=0
MOVL C02011 V=800.0 PL=0
MOVL C02012 V=800.0 PL=0
MOVL C02013 V=800.0 PL=0
MOVL C02014 V=800.0 PL=0
MOVL C02015 V=800.0 PL=0
MOVL C02016 V=800.0 PL=0
MOVL C02017 V=800.0 PL=0
MOVL C02018 V=800.0 PL=0
MOVL C02019 V=800.0 PL=0
MOVL C02020 V=800.0 PL=0
MOVL C02021 V=800.0 PL=0
MOVL C02022 V=800.0 PL=0
MOVL C02023 V=800.0 PL=0
MOVL C02024 V=800.0 PL=0
MOVL C02025 V=800.0 PL=0
MOVL C02026 V=800.0 PL=0
MOVL C02027 V=800.0 PL=0
MOVL C02028 V=800.0 PL=0
MOVL C02029 V=800.0 PL=0
MOVL C02030 V=800.0 PL=0
MOVL C02031 V=800.0 PL=0
MOVL C02032 V=800.0 PL=0
MOVL C02033 V=800.0 PL=0
MOVL C02034 V=800.0 PL=0
MOVL C02035 V=800.0 PL=0
MOVL C02036 V=800.0 PL=0
MOVL C02037 V=800.0 PL=0
MOVL C02038 V=800.0 PL=0
MOVL C02039 V=800.0 PL=0
MOVL C02040 V=800.0 PL=0
MOVL C02041 V=800.0 PL=0
MOVL C02042 V=800.0 PL=0
MOVL C02043 V=800.0 PL=0
MOVL C02044 V=800.0 PL=0
MOVL C02045 V=800.0 PL=0
MOVL C02046 V=800.0 PL=0
MOVL C02047 V=800.0 PL=0
MOVL C02048 V=800.0 PL=0
MOVL C02049 V=800.0 PL=0
MOVL C02050 V=800.0 PL=0
MOVL C02051 V=800.0 PL=0
MOVL C02052 V=800.0 PL=0
MOVL C02053 V=800.0 PL=0
MOVL C02054 V=800.0 PL=0
MOVL C02055 V=800.0 PL=0
MOVL C02056 V=800.0 PL=0
MOVL C02057 V=800.0 PL=0
MOVL C02058 V=800.0 PL=0
MOVL C02059 V=800.0 PL=0
MOVL C02060 V=800.0 PL=0
MOVL C02061 V=800.0 PL=0
MOVL C02062 V=800.0 PL=0
MOVL C02063 V=800.0 PL=0
MOVL C02064 V=800.0 PL=0
MOVL C02065 V=800.0 PL=0
MOVL C02066 V=800.0 PL=0
MOVL C02067 V=800.0 PL=0
MOVL C02068 V=800.0 PL=0
MOVL C02069 V=800.0 PL=0
MOVL C02070 V=800.0 PL=0
MOVL C02071 V=800.0 PL=0
MOVL C02072 V=800.0 PL=0
MOVL C02073 V=800.0 PL=0
MOVL C02074 V=800.0 PL=0
MOVL C02075 V=800.0 PL=0
MOVL C02076 V=800.0 PL=0
MOVL C02077 V=800.0 PL=0
MOVL C02078 V=800.0 PL=0
MOVL C02079 V=800.0 PL=0
MOVL C02080 V=800.0 PL=0
MOVL C02081 V=800.0 PL=0
MOVL C02082 V=800.0 PL=0
MOVL C02083 V=800.0 PL=0
MOVL C02084 V=800.0 PL=0
MOVL C02085 V=800.0 PL=0
MOVL C02086 V=800.0 PL=0
MOVL C02087 V=800.0 PL=0
MOVL C02088 V=800.0 PL=0
MOVL C02089 V=800.0 PL=0
MOVL C02090 V=800.0 PL=0
MOVL C02091 V=800.0 PL=0
MOVL C02092 V=800.0 PL=0
MOVL C02093 V=800.0 PL=0
MOVL C02094 V=800.0 PL=0
MOVL C02095 V=800.0 PL=0
MOVL C02096 V=800.0 PL=0
MOVL C02097 V=800.0 PL=0
MOVL C02098 V=800.0 PL=0
MOVL C02099 V=800.0 PL=0
MOVL C02100 V=800.0 PL=0
